LIN {X 0,Y 363.86,Z 414.069,A -85,B 0,C 180,E1 -13028.68,E2 -13028.68} C_VEL
LIN {X 0,Y 368.612,Z 450.307,A -85,B 0,C 180,E1 -13029.654,E2 -13029.654} C_VEL
LIN {X 0,Y 367.486,Z 523.043,A -85,B 0,C 180,E1 -13031.1,E2 -13031.1} C_VEL
LIN {X 0,Y 366.851,Z 536.983,A -85,B 0,C 180,E1 -13031.609,E2 -13031.609} C_VEL
LIN {X 0,Y 366.037,Z 549.991,A -85,B 0,C 180,E1 -13032.326,E2 -13032.326} C_VEL
LIN {X 0,Y 365.038,Z 561.815,A -85,B 0,C 180,E1 -13033.215,E2 -13033.215} C_VEL
LIN {X 0,Y 364.036,Z 573.232,A -85,B 0,C 180,E1 -13034.319,E2 -13034.319} C_VEL
LIN {X 0,Y 363.244,Z 583.53,A -85,B 0,C 180,E1 -13035.576,E2 -13035.576} C_VEL
LIN {X 0,Y 362.317,Z 593.595,A -85,B 0,C 180,E1 -13037.111,E2 -13037.111} C_VEL
LIN {X 0,Y 361.455,Z 602.44,A -85,B 0,C 180,E1 -13038.788,E2 -13038.788} C_VEL
LIN {X 0,Y 360.952,Z 609.493,A -85,B 0,C 180,E1 -13040.474,E2 -13040.474} C_VEL
LIN {X 0,Y 360.641,Z 615.132,A -85,B 0,C 180,E1 -13042.16,E2 -13042.16} C_VEL
LIN {X 0,Y 360.454,Z 619.728,A -85,B 0,C 180,E1 -13043.923,E2 -13043.923} C_VEL
LIN {X 0,Y 360.429,Z 622.876,A -85,B 0,C 180,E1 -13045.527,E2 -13045.527} C_VEL
LIN {X 0,Y 360.392,Z 625.76,A -85,B 0,C 180,E1 -13047.765,E2 -13047.765} C_VEL
LIN {X 0,Y 360.474,Z 626.578,A -85,B 0,C 180,E1 -13048.883,E2 -13048.883} C_VEL
LIN {X 0,Y 360.477,Z 626.96,A -85,B 0,C 180,E1 -13050,E2 -13050} C_VEL
LIN {X 0,Y 360.453,Z 626.953,A -85,B 0,C 180,E1 -13051.117,E2 -13051.117} C_VEL
LIN {X 0,Y 360.352,Z 626.554,A -85,B 0,C 180,E1 -13052.235,E2 -13052.235} C_VEL
LIN {X 0,Y 360.326,Z 625.757,A -85,B 0,C 180,E1 -13053.354,E2 -13053.354} C_VEL
LIN {X 0,Y 360.371,Z 624.522,A -85,B 0,C 180,E1 -13054.474,E2 -13054.474} C_VEL
LIN {X 0,Y 360.435,Z 622.125,A -85,B 0,C 180,E1 -13056.048,E2 -13056.048} C_VEL
LIN {X 0,Y 360.659,Z 618.313,A -85,B 0,C 180,E1 -13057.84,E2 -13057.84} C_VEL
LIN {X 0,Y 361.038,Z 613.617,A -85,B 0,C 180,E1 -13059.524,E2 -13059.524} C_VEL
LIN {X 0,Y 361.792,Z 606.572,A -85,B 0,C 180,E1 -13061.485,E2 -13061.485} C_VEL
LIN {X 0,Y 362.814,Z 598.979,A -85,B 0,C 180,E1 -13063.156,E2 -13063.156} C_VEL
LIN {X 0,Y 363.882,Z 589.935,A -85,B 0,C 180,E1 -13064.755,E2 -13064.755} C_VEL
LIN {X 0,Y 365.122,Z 579.71,A -85,B 0,C 180,E1 -13066.206,E2 -13066.206} C_VEL
LIN {X 0,Y 366.496,Z 568.849,A -85,B 0,C 180,E1 -13067.435,E2 -13067.435} C_VEL
LIN {X 0,Y 367.703,Z 558.247,A -85,B 0,C 180,E1 -13068.383,E2 -13068.383} C_VEL
LIN {X 0,Y 368.961,Z 545.524,A -85,B 0,C 180,E1 -13069.254,E2 -13069.254} C_VEL
LIN {X 0,Y 369.904,Z 532.782,A -85,B 0,C 180,E1 -13069.889,E2 -13069.889} C_VEL
LIN {X 0,Y 370.533,Z 519.302,A -85,B 0,C 180,E1 -13070.316,E2 -13070.316} C_VEL
LIN {X 0,Y 371.83,Z 449.639,A -85,B 0,C 180,E1 -13071.708,E2 -13071.708} C_VEL
LIN {X 0,Y 368.724,Z 429.89,A -85,B 0,C 180,E1 -13072.358,E2 -13072.358} C_VEL
LIN {X 0,Y 365.446,Z 413.267,A -85,B 0,C 180,E1 -13072.99,E2 -13072.99} C_VEL
LIN {X 0,Y 366.949,Z 399.466,A -85,B 0,C 180,E1 -13076.136,E2 -13076.136} C_VEL
LIN {X 0,Y 365.22,Z 390.34,A -85,B 0,C 180,E1 -13078.493,E2 -13078.493} C_VEL
LIN {X 0,Y 362.261,Z 377.933,A -85,B 0,C 180,E1 -13081.914,E2 -13081.914} C_VEL
LIN {X 0,Y 361.88,Z 376.409,A -85,B 0,C 180,E1 -13082.362,E2 -13082.362} C_VEL
LIN {X 0,Y 361.866,Z 376.411,A -85,B 0,C 180,E1 -13085.636,E2 -13085.636} C_VEL
LIN {X 0,Y 361.872,Z 376.403,A -85,B 0,C 180,E1 -13089.027,E2 -13089.027} C_VEL
LIN {X 0,Y 361.854,Z 376.402,A -85,B 0,C 180,E1 -13092.435,E2 -13092.435} C_VEL
LIN {X 0,Y 361.908,Z 376.405,A -85,B 0,C 180,E1 -13095.93,E2 -13095.93} C_VEL
LIN {X 0,Y 361.901,Z 376.405,A -85,B 0,C 180,E1 -13099.231,E2 -13099.231} C_VEL
LIN {X 0,Y 361.864,Z 376.405,A -85,B 0,C 180,E1 -13102.982,E2 -13102.982} C_VEL
LIN {X 0,Y 361.853,Z 376.404,A -85,B 0,C 180,E1 -13106.63,E2 -13106.63} C_VEL
LIN {X 0,Y 361.87,Z 376.404,A -85,B 0,C 180,E1 -13109.672,E2 -13109.672} C_VEL
LIN {X 0,Y 361.948,Z 376.394,A -85,B 0,C 180,E1 -13113.475,E2 -13113.475} C_VEL
LIN {X 0,Y 361.883,Z 376.406,A -85,B 0,C 180,E1 -13117.144,E2 -13117.144} C_VEL
LIN {X 0,Y 361.913,Z 376.402,A -85,B 0,C 180,E1 -13120.724,E2 -13120.724} C_VEL
LIN {X 0,Y 361.94,Z 376.398,A -85,B 0,C 180,E1 -13124.226,E2 -13124.226} C_VEL
LIN {X 0,Y 361.991,Z 376.389,A -85,B 0,C 180,E1 -13126.528,E2 -13126.528} C_VEL
LIN {X 0,Y 362.023,Z 376.389,A -85,B 0,C 180,E1 -13129.938,E2 -13129.938} C_VEL
LIN {X 0,Y 362.155,Z 376.365,A -85,B 0,C 180,E1 -13133.314,E2 -13133.314} C_VEL
LIN {X 0,Y 362.275,Z 376.35,A -85,B 0,C 180,E1 -13137.777,E2 -13137.777} C_VEL
LIN {X 0,Y 362.422,Z 376.339,A -85,B 0,C 180,E1 -13140,E2 -13140} C_VEL
LIN {X 0,Y 362.276,Z 376.348,A -85,B 0,C 180,E1 -13142.224,E2 -13142.224} C_VEL
LIN {X 0,Y 362.157,Z 376.369,A -85,B 0,C 180,E1 -13146.687,E2 -13146.687} C_VEL
LIN {X 0,Y 362.024,Z 376.388,A -85,B 0,C 180,E1 -13150.063,E2 -13150.063} C_VEL
LIN {X 0,Y 361.991,Z 376.393,A -85,B 0,C 180,E1 -13153.899,E2 -13153.899} C_VEL
LIN {X 0,Y 361.962,Z 376.396,A -85,B 0,C 180,E1 -13157.94,E2 -13157.94} C_VEL
LIN {X 0,Y 361.906,Z 376.404,A -85,B 0,C 180,E1 -13161.652,E2 -13161.652} C_VEL
LIN {X 0,Y 361.923,Z 376.404,A -85,B 0,C 180,E1 -13165.291,E2 -13165.291} C_VEL
LIN {X 0,Y 361.903,Z 376.402,A -85,B 0,C 180,E1 -13167.78,E2 -13167.78} C_VEL
LIN {X 0,Y 361.833,Z 376.414,A -85,B 0,C 180,E1 -13171.63,E2 -13171.63} C_VEL
LIN {X 0,Y 361.871,Z 376.401,A -85,B 0,C 180,E1 -13175.346,E2 -13175.346} C_VEL
LIN {X 0,Y 361.872,Z 376.41,A -85,B 0,C 180,E1 -13179.029,E2 -13179.029} C_VEL
LIN {X 0,Y 361.882,Z 376.4,A -85,B 0,C 180,E1 -13182.441,E2 -13182.441} C_VEL
LIN {X 0,Y 361.846,Z 376.409,A -85,B 0,C 180,E1 -13185.637,E2 -13185.637} C_VEL
LIN {X 0,Y 361.873,Z 376.574,A -85,B 0,C 180,E1 -13188.55,E2 -13188.55} C_VEL
LIN {X 0,Y 363.569,Z 383.949,A -85,B 0,C 180,E1 -13190.931,E2 -13190.931} C_VEL
LIN {X 0,Y 371.29,Z 402.274,A -85,B 0,C 180,E1 -13191.936,E2 -13191.936} C_VEL
LIN {X 0,Y 372.737,Z 408.261,A -85,B 0,C 180,E1 -13192.173,E2 -13192.173} C_VEL
LIN {X 0,Y 370.929,Z 490.598,A -85,B 0,C 180,E1 -13193.821,E2 -13193.821} C_VEL
LIN {X 0,Y 370.307,Z 504.489,A -85,B 0,C 180,E1 -13194.342,E2 -13194.342} C_VEL
LIN {X 0,Y 369.584,Z 516.079,A -85,B 0,C 180,E1 -13194.985,E2 -13194.985} C_VEL
LIN {X 0,Y 368.499,Z 528.657,A -85,B 0,C 180,E1 -13195.929,E2 -13195.929} C_VEL
LIN {X 0,Y 367.416,Z 539.356,A -85,B 0,C 180,E1 -13196.966,E2 -13196.966} C_VEL
LIN {X 0,Y 366.121,Z 550.319,A -85,B 0,C 180,E1 -13198.3,E2 -13198.3} C_VEL
LIN {X 0,Y 364.993,Z 559.126,A -85,B 0,C 180,E1 -13199.64,E2 -13199.64} C_VEL
LIN {X 0,Y 363.917,Z 567.14,A -85,B 0,C 180,E1 -13201.132,E2 -13201.132} C_VEL
LIN {X 0,Y 362.952,Z 574.158,A -85,B 0,C 180,E1 -13202.74,E2 -13202.74} C_VEL
LIN {X 0,Y 362.27,Z 579.094,A -85,B 0,C 180,E1 -13204.12,E2 -13204.12} C_VEL
LIN {X 0,Y 361.543,Z 584.472,A -85,B 0,C 180,E1 -13206.013,E2 -13206.013} C_VEL
LIN {X 0,Y 361.041,Z 588.073,A -85,B 0,C 180,E1 -13207.693,E2 -13207.693} C_VEL
LIN {X 0,Y 360.706,Z 590.795,A -85,B 0,C 180,E1 -13209.47,E2 -13209.47} C_VEL
LIN {X 0,Y 360.459,Z 592.046,A -85,B 0,C 180,E1 -13210.643,E2 -13210.643} C_VEL
LIN {X 0,Y 360.346,Z 592.816,A -85,B 0,C 180,E1 -13211.817,E2 -13211.817} C_VEL
LIN {X 0,Y 360.319,Z 593.156,A -85,B 0,C 180,E1 -13212.988,E2 -13212.988} C_VEL
LIN {X 0,Y 360.266,Z 593.094,A -85,B 0,C 180,E1 -13214.151,E2 -13214.151} C_VEL
LIN {X 0,Y 360.268,Z 592.604,A -85,B 0,C 180,E1 -13215.31,E2 -13215.31} C_VEL
LIN {X 0,Y 360.406,Z 590.903,A -85,B 0,C 180,E1 -13217.167,E2 -13217.167} C_VEL
LIN {X 0,Y 360.694,Z 587.473,A -85,B 0,C 180,E1 -13219.333,E2 -13219.333} C_VEL
LIN {X 0,Y 360.984,Z 583.589,A -85,B 0,C 180,E1 -13221.04,E2 -13221.04} C_VEL
LIN {X 0,Y 361.463,Z 578.015,A -85,B 0,C 180,E1 -13222.905,E2 -13222.905} C_VEL
LIN {X 0,Y 362.051,Z 571.018,A -85,B 0,C 180,E1 -13224.71,E2 -13224.71} C_VEL
LIN {X 0,Y 362.839,Z 562.825,A -85,B 0,C 180,E1 -13226.391,E2 -13226.391} C_VEL
LIN {X 0,Y 363.609,Z 554.46,A -85,B 0,C 180,E1 -13227.785,E2 -13227.785} C_VEL
LIN {X 0,Y 364.602,Z 544.132,A -85,B 0,C 180,E1 -13229.172,E2 -13229.172} C_VEL
LIN {X 0,Y 365.465,Z 533.637,A -85,B 0,C 180,E1 -13230.303,E2 -13230.303} C_VEL
LIN {X 0,Y 366.263,Z 522.766,A -85,B 0,C 180,E1 -13231.237,E2 -13231.237} C_VEL
LIN {X 0,Y 367.003,Z 510.308,A -85,B 0,C 180,E1 -13232.058,E2 -13232.058} C_VEL
LIN {X 0,Y 367.525,Z 497.927,A -85,B 0,C 180,E1 -13232.637,E2 -13232.637} C_VEL
LIN {X 0,Y 367.83,Z 485.609,A -85,B 0,C 180,E1 -13233.012,E2 -13233.012} C_VEL
LIN {X 0,Y 369.047,Z 405.84,A -85,B 0,C 180,E1 -13234.574,E2 -13234.574} C_VEL
LIN {X 0,Y 366.205,Z 392.374,A -85,B 0,C 180,E1 -13234.989,E2 -13234.989} C_VEL
LIN {X 0,Y 363.231,Z 382.868,A -85,B 0,C 180,E1 -13235.365,E2 -13235.365} C_VEL
LIN {X 0,Y 362.665,Z 379.195,A -85,B 0,C 180,E1 -13236.426,E2 -13236.426} C_VEL
LIN {X 0,Y 362.058,Z 377.775,A -85,B 0,C 180,E1 -13236.985,E2 -13236.985} C_VEL
LIN {X 0,Y 361.037,Z 377.05,A -85,B 0,C 180,E1 -13237.568,E2 -13237.568} C_VEL
LIN {X 0,Y 358.444,Z 376.838,A -85,B 0,C 180,E1 -13238.759,E2 -13238.759} C_VEL
LIN {X 0,Y 356.003,Z 377.137,A -85,B 0,C 180,E1 -13240.005,E2 -13240.005} C_VEL
LIN {X 0,Y 355.005,Z 377.264,A -85,B 0,C 180,E1 -13240.97,E2 -13240.97} C_VEL
LIN {X 0,Y 354.935,Z 377.274,A -85,B 0,C 180,E1 -13241.296,E2 -13241.296} C_VEL
LIN {X 0,Y 354.924,Z 377.273,A -85,B 0,C 180,E1 -13244.917,E2 -13244.917} C_VEL
LIN {X 0,Y 354.905,Z 377.273,A -85,B 0,C 180,E1 -13248.471,E2 -13248.471} C_VEL
LIN {X 0,Y 354.839,Z 377.281,A -85,B 0,C 180,E1 -13252.105,E2 -13252.105} C_VEL
LIN {X 0,Y 354.902,Z 377.274,A -85,B 0,C 180,E1 -13255.827,E2 -13255.827} C_VEL
LIN {X 0,Y 354.856,Z 377.281,A -85,B 0,C 180,E1 -13259.678,E2 -13259.678} C_VEL
LIN {X 0,Y 354.807,Z 377.286,A -85,B 0,C 180,E1 -13263.701,E2 -13263.701} C_VEL
LIN {X 0,Y 354.799,Z 377.287,A -85,B 0,C 180,E1 -13266.458,E2 -13266.458} C_VEL
LIN {X 0,Y 354.824,Z 377.286,A -85,B 0,C 180,E1 -13269.423,E2 -13269.423} C_VEL
LIN {X 0,Y 354.787,Z 377.292,A -85,B 0,C 180,E1 -13272.866,E2 -13272.866} C_VEL
LIN {X 0,Y 354.774,Z 377.289,A -85,B 0,C 180,E1 -13276.104,E2 -13276.104} C_VEL
LIN {X 0,Y 354.787,Z 377.292,A -85,B 0,C 180,E1 -13279.178,E2 -13279.178} C_VEL
LIN {X 0,Y 354.805,Z 377.287,A -85,B 0,C 180,E1 -13282.401,E2 -13282.401} C_VEL
LIN {X 0,Y 354.809,Z 377.291,A -85,B 0,C 180,E1 -13284.94,E2 -13284.94} C_VEL
LIN {X 0,Y 354.789,Z 377.289,A -85,B 0,C 180,E1 -13288.404,E2 -13288.404} C_VEL
LIN {X 0,Y 354.841,Z 377.281,A -85,B 0,C 180,E1 -13291.618,E2 -13291.618} C_VEL
LIN {X 0,Y 354.894,Z 377.275,A -85,B 0,C 180,E1 -13294.172,E2 -13294.172} C_VEL
LIN {X 0,Y 354.829,Z 377.283,A -85,B 0,C 180,E1 -13297.893,E2 -13297.893} C_VEL
LIN {X 0,Y 354.916,Z 377.272,A -85,B 0,C 180,E1 -13301.891,E2 -13301.891} C_VEL
LIN {X 0,Y 354.936,Z 377.27,A -85,B 0,C 180,E1 -13305.981,E2 -13305.981} C_VEL
LIN {X 0,Y 354.971,Z 377.265,A -85,B 0,C 180,E1 -13309.735,E2 -13309.735} C_VEL
LIN {X 0,Y 355.119,Z 377.247,A -85,B 0,C 180,E1 -13313.18,E2 -13313.18} C_VEL
LIN {X 0,Y 355.238,Z 377.232,A -85,B 0,C 180,E1 -13317.732,E2 -13317.732} C_VEL
LIN {X 0,Y 355.389,Z 377.214,A -85,B 0,C 180,E1 -13320,E2 -13320} C_VEL
LIN {X 0,Y 355.238,Z 377.235,A -85,B 0,C 180,E1 -13322.267,E2 -13322.267} C_VEL
LIN {X 0,Y 355.118,Z 377.249,A -85,B 0,C 180,E1 -13326.819,E2 -13326.819} C_VEL
LIN {X 0,Y 354.97,Z 377.27,A -85,B 0,C 180,E1 -13330.264,E2 -13330.264} C_VEL
LIN {X 0,Y 354.935,Z 377.272,A -85,B 0,C 180,E1 -13334.019,E2 -13334.019} C_VEL
LIN {X 0,Y 354.915,Z 377.276,A -85,B 0,C 180,E1 -13338.109,E2 -13338.109} C_VEL
LIN {X 0,Y 354.827,Z 377.287,A -85,B 0,C 180,E1 -13342.106,E2 -13342.106} C_VEL
LIN {X 0,Y 354.893,Z 377.277,A -85,B 0,C 180,E1 -13345.828,E2 -13345.828} C_VEL
LIN {X 0,Y 354.848,Z 377.282,A -85,B 0,C 180,E1 -13349.679,E2 -13349.679} C_VEL
LIN {X 0,Y 354.8,Z 377.288,A -85,B 0,C 180,E1 -13353.703,E2 -13353.703} C_VEL
LIN {X 0,Y 354.794,Z 377.29,A -85,B 0,C 180,E1 -13356.46,E2 -13356.46} C_VEL
LIN {X 0,Y 354.819,Z 377.284,A -85,B 0,C 180,E1 -13359.424,E2 -13359.424} C_VEL
LIN {X 0,Y 354.833,Z 377.282,A -85,B 0,C 180,E1 -13362.877,E2 -13362.877} C_VEL
LIN {X 0,Y 354.801,Z 377.291,A -85,B 0,C 180,E1 -13366.11,E2 -13366.11} C_VEL
LIN {X 0,Y 354.821,Z 377.284,A -85,B 0,C 180,E1 -13369.185,E2 -13369.185} C_VEL
LIN {X 0,Y 354.807,Z 377.287,A -85,B 0,C 180,E1 -13372.403,E2 -13372.403} C_VEL
LIN {X 0,Y 354.811,Z 377.285,A -85,B 0,C 180,E1 -13374.942,E2 -13374.942} C_VEL
LIN {X 0,Y 354.814,Z 377.286,A -85,B 0,C 180,E1 -13378.4,E2 -13378.4} C_VEL
LIN {X 0,Y 354.873,Z 377.309,A -85,B 0,C 180,E1 -13379.751,E2 -13379.751} C_VEL
LIN {X 0,Y 357.344,Z 389.276,A -85,B 0,C 180,E1 -13382.74,E2 -13382.74} C_VEL
LIN {X 0,Y 358.518,Z 396.396,A -85,B 0,C 180,E1 -13384.453,E2 -13384.453} C_VEL
LIN {X 0,Y 357.215,Z 410.591,A -85,B 0,C 180,E1 -13387.623,E2 -13387.623} C_VEL
LIN {X 0,Y 356.949,Z 413.959,A -85,B 0,C 180,E1 -13388.339,E2 -13388.339} C_VEL
LIN {X 0,Y 361.826,Z 449.698,A -85,B 0,C 180,E1 -13389.323,E2 -13389.323} C_VEL
LIN {X 0,Y 360.656,Z 522.733,A -85,B 0,C 180,E1 -13390.802,E2 -13390.802} C_VEL
LIN {X 0,Y 359.983,Z 536.659,A -85,B 0,C 180,E1 -13391.319,E2 -13391.319} C_VEL
LIN {X 0,Y 359.162,Z 549.668,A -85,B 0,C 180,E1 -13392.05,E2 -13392.05} C_VEL
LIN {X 0,Y 358.052,Z 562.287,A -85,B 0,C 180,E1 -13393.024,E2 -13393.024} C_VEL
LIN {X 0,Y 357.031,Z 573.556,A -85,B 0,C 180,E1 -13394.15,E2 -13394.15} C_VEL
LIN {X 0,Y 356.157,Z 584.466,A -85,B 0,C 180,E1 -13395.542,E2 -13395.542} C_VEL
LIN {X 0,Y 355.307,Z 592.85,A -85,B 0,C 180,E1 -13396.852,E2 -13396.852} C_VEL
LIN {X 0,Y 354.454,Z 601.776,A -85,B 0,C 180,E1 -13398.564,E2 -13398.564} C_VEL
LIN {X 0,Y 353.924,Z 608.914,A -85,B 0,C 180,E1 -13400.283,E2 -13400.283} C_VEL
LIN {X 0,Y 353.565,Z 614.604,A -85,B 0,C 180,E1 -13402.002,E2 -13402.002} C_VEL
LIN {X 0,Y 353.368,Z 619.576,A -85,B 0,C 180,E1 -13403.951,E2 -13403.951} C_VEL
LIN {X 0,Y 353.338,Z 622.437,A -85,B 0,C 180,E1 -13405.437,E2 -13405.437} C_VEL
LIN {X 0,Y 353.295,Z 625.36,A -85,B 0,C 180,E1 -13407.72,E2 -13407.72} C_VEL
LIN {X 0,Y 353.392,Z 626.212,A -85,B 0,C 180,E1 -13408.86,E2 -13408.86} C_VEL
LIN {X 0,Y 353.395,Z 626.617,A -85,B 0,C 180,E1 -13410,E2 -13410} C_VEL
LIN {X 0,Y 353.355,Z 626.626,A -85,B 0,C 180,E1 -13411.14,E2 -13411.14} C_VEL
LIN {X 0,Y 353.246,Z 625.479,A -85,B 0,C 180,E1 -13413.422,E2 -13413.422} C_VEL
LIN {X 0,Y 353.284,Z 624.273,A -85,B 0,C 180,E1 -13414.564,E2 -13414.564} C_VEL
LIN {X 0,Y 353.328,Z 622.209,A -85,B 0,C 180,E1 -13415.987,E2 -13415.987} C_VEL
LIN {X 0,Y 353.605,Z 618.147,A -85,B 0,C 180,E1 -13417.997,E2 -13417.997} C_VEL
LIN {X 0,Y 354.006,Z 613.497,A -85,B 0,C 180,E1 -13419.715,E2 -13419.715} C_VEL
LIN {X 0,Y 354.824,Z 606.503,A -85,B 0,C 180,E1 -13421.713,E2 -13421.713} C_VEL
LIN {X 0,Y 355.896,Z 598.967,A -85,B 0,C 180,E1 -13423.416,E2 -13423.416} C_VEL
LIN {X 0,Y 356.96,Z 590.321,A -85,B 0,C 180,E1 -13424.999,E2 -13424.999} C_VEL
LIN {X 0,Y 358.304,Z 579.889,A -85,B 0,C 180,E1 -13426.523,E2 -13426.523} C_VEL
LIN {X 0,Y 359.758,Z 569.166,A -85,B 0,C 180,E1 -13427.772,E2 -13427.772} C_VEL
LIN {X 0,Y 361.014,Z 558.779,A -85,B 0,C 180,E1 -13428.736,E2 -13428.736} C_VEL
LIN {X 0,Y 362.286,Z 546.334,A -85,B 0,C 180,E1 -13429.624,E2 -13429.624} C_VEL
LIN {X 0,Y 363.328,Z 533.266,A -85,B 0,C 180,E1 -13430.302,E2 -13430.302} C_VEL
LIN {X 0,Y 364.03,Z 520.256,A -85,B 0,C 180,E1 -13430.741,E2 -13430.741} C_VEL
LIN {X 0,Y 365.417,Z 450.753,A -85,B 0,C 180,E1 -13432.157,E2 -13432.157} C_VEL
LIN {X 0,Y 362.436,Z 431.394,A -85,B 0,C 180,E1 -13432.808,E2 -13432.808} C_VEL
LIN {X 0,Y 358.762,Z 412.874,A -85,B 0,C 180,E1 -13433.539,E2 -13433.539} C_VEL
LIN {X 0,Y 360.085,Z 401.05,A -85,B 0,C 180,E1 -13436.298,E2 -13436.298} C_VEL
LIN {X 0,Y 358.348,Z 391.895,A -85,B 0,C 180,E1 -13438.717,E2 -13438.717} C_VEL
LIN {X 0,Y 355.341,Z 379.317,A -85,B 0,C 180,E1 -13442.276,E2 -13442.276} C_VEL
LIN {X 0,Y 354.831,Z 377.283,A -85,B 0,C 180,E1 -13442.918,E2 -13442.918} C_VEL
LIN {X 0,Y 354.8,Z 377.291,A -85,B 0,C 180,E1 -13446.458,E2 -13446.458} C_VEL
LIN {X 0,Y 354.821,Z 377.284,A -85,B 0,C 180,E1 -13449.423,E2 -13449.423} C_VEL
LIN {X 0,Y 354.804,Z 377.283,A -85,B 0,C 180,E1 -13452.87,E2 -13452.87} C_VEL
LIN {X 0,Y 354.848,Z 377.286,A -85,B 0,C 180,E1 -13456.116,E2 -13456.116} C_VEL
LIN {X 0,Y 354.852,Z 377.283,A -85,B 0,C 180,E1 -13459.188,E2 -13459.188} C_VEL
LIN {X 0,Y 354.804,Z 377.286,A -85,B 0,C 180,E1 -13462.402,E2 -13462.402} C_VEL
LIN {X 0,Y 354.807,Z 377.287,A -85,B 0,C 180,E1 -13464.94,E2 -13464.94} C_VEL
LIN {X 0,Y 354.788,Z 377.289,A -85,B 0,C 180,E1 -13468.405,E2 -13468.405} C_VEL
LIN {X 0,Y 354.847,Z 377.283,A -85,B 0,C 180,E1 -13471.619,E2 -13471.619} C_VEL
LIN {X 0,Y 354.893,Z 377.271,A -85,B 0,C 180,E1 -13474.172,E2 -13474.172} C_VEL
LIN {X 0,Y 354.827,Z 377.278,A -85,B 0,C 180,E1 -13477.894,E2 -13477.894} C_VEL
LIN {X 0,Y 354.916,Z 377.268,A -85,B 0,C 180,E1 -13481.891,E2 -13481.891} C_VEL
LIN {X 0,Y 354.935,Z 377.27,A -85,B 0,C 180,E1 -13485.981,E2 -13485.981} C_VEL
LIN {X 0,Y 354.97,Z 377.27,A -85,B 0,C 180,E1 -13489.736,E2 -13489.736} C_VEL
LIN {X 0,Y 355.119,Z 377.24,A -85,B 0,C 180,E1 -13493.181,E2 -13493.181} C_VEL
LIN {X 0,Y 355.238,Z 377.226,A -85,B 0,C 180,E1 -13497.733,E2 -13497.733} C_VEL
LIN {X 0,Y 355.391,Z 377.215,A -85,B 0,C 180,E1 -13500,E2 -13500} C_VEL
LIN {X 0,Y 355.239,Z 377.224,A -85,B 0,C 180,E1 -13502.268,E2 -13502.268} C_VEL
LIN {X 0,Y 355.12,Z 377.244,A -85,B 0,C 180,E1 -13506.82,E2 -13506.82} C_VEL
LIN {X 0,Y 354.971,Z 377.266,A -85,B 0,C 180,E1 -13510.265,E2 -13510.265} C_VEL
LIN {X 0,Y 354.936,Z 377.271,A -85,B 0,C 180,E1 -13514.019,E2 -13514.019} C_VEL
LIN {X 0,Y 354.917,Z 377.273,A -85,B 0,C 180,E1 -13518.11,E2 -13518.11} C_VEL
LIN {X 0,Y 354.841,Z 377.283,A -85,B 0,C 180,E1 -13522.106,E2 -13522.106} C_VEL
LIN {X 0,Y 354.894,Z 377.277,A -85,B 0,C 180,E1 -13525.828,E2 -13525.828} C_VEL
LIN {X 0,Y 354.813,Z 377.285,A -85,B 0,C 180,E1 -13529.683,E2 -13529.683} C_VEL
LIN {X 0,Y 354.802,Z 377.277,A -85,B 0,C 180,E1 -13533.703,E2 -13533.703} C_VEL
LIN {X 0,Y 354.796,Z 377.291,A -85,B 0,C 180,E1 -13536.46,E2 -13536.46} C_VEL
LIN {X 0,Y 354.821,Z 377.285,A -85,B 0,C 180,E1 -13539.425,E2 -13539.425} C_VEL
LIN {X 0,Y 354.833,Z 377.281,A -85,B 0,C 180,E1 -13542.876,E2 -13542.876} C_VEL
LIN {X 0,Y 354.783,Z 377.293,A -85,B 0,C 180,E1 -13546.107,E2 -13546.107} C_VEL
LIN {X 0,Y 354.814,Z 377.389,A -85,B 0,C 180,E1 -13548.045,E2 -13548.045} C_VEL
LIN {X 0,Y 356.388,Z 384.235,A -85,B 0,C 180,E1 -13550.335,E2 -13550.335} C_VEL
LIN {X 0,Y 364.963,Z 404.134,A -85,B 0,C 180,E1 -13551.486,E2 -13551.486} C_VEL
LIN {X 0,Y 366.344,Z 409.497,A -85,B 0,C 180,E1 -13551.711,E2 -13551.711} C_VEL
LIN {X 0,Y 364.451,Z 491.149,A -85,B 0,C 180,E1 -13553.375,E2 -13553.375} C_VEL
LIN {X 0,Y 363.826,Z 504.929,A -85,B 0,C 180,E1 -13553.904,E2 -13553.904} C_VEL
LIN {X 0,Y 363.019,Z 516.869,A -85,B 0,C 180,E1 -13554.58,E2 -13554.58} C_VEL
LIN {X 0,Y 362.046,Z 527.796,A -85,B 0,C 180,E1 -13555.404,E2 -13555.404} C_VEL
LIN {X 0,Y 360.896,Z 538.696,A -85,B 0,C 180,E1 -13556.458,E2 -13556.458} C_VEL
LIN {X 0,Y 359.499,Z 549.854,A -85,B 0,C 180,E1 -13557.814,E2 -13557.814} C_VEL
LIN {X 0,Y 358.207,Z 559.688,A -85,B 0,C 180,E1 -13559.329,E2 -13559.329} C_VEL
LIN {X 0,Y 357.055,Z 567.654,A -85,B 0,C 180,E1 -13560.847,E2 -13560.847} C_VEL
LIN {X 0,Y 355.899,Z 575.485,A -85,B 0,C 180,E1 -13562.702,E2 -13562.702} C_VEL
LIN {X 0,Y 355.183,Z 580.498,A -85,B 0,C 180,E1 -13564.195,E2 -13564.195} C_VEL
LIN {X 0,Y 354.551,Z 584.755,A -85,B 0,C 180,E1 -13565.76,E2 -13565.76} C_VEL
LIN {X 0,Y 353.934,Z 589.029,A -85,B 0,C 180,E1 -13567.835,E2 -13567.835} C_VEL
LIN {X 0,Y 353.679,Z 590.826,A -85,B 0,C 180,E1 -13569.06,E2 -13569.06} C_VEL
LIN {X 0,Y 353.462,Z 592.131,A -85,B 0,C 180,E1 -13570.244,E2 -13570.244} C_VEL
LIN {X 0,Y 353.287,Z 593.034,A -85,B 0,C 180,E1 -13571.441,E2 -13571.441} C_VEL
LIN {X 0,Y 353.211,Z 593.478,A -85,B 0,C 180,E1 -13572.763,E2 -13572.763} C_VEL
LIN {X 0,Y 353.18,Z 593.076,A -85,B 0,C 180,E1 -13575.008,E2 -13575.008} C_VEL
LIN {X 0,Y 353.299,Z 591.322,A -85,B 0,C 180,E1 -13577.095,E2 -13577.095} C_VEL
LIN {X 0,Y 353.56,Z 588.282,A -85,B 0,C 180,E1 -13579.115,E2 -13579.115} C_VEL
LIN {X 0,Y 353.854,Z 584.552,A -85,B 0,C 180,E1 -13580.858,E2 -13580.858} C_VEL
LIN {X 0,Y 354.295,Z 579.422,A -85,B 0,C 180,E1 -13582.675,E2 -13582.675} C_VEL
LIN {X 0,Y 354.938,Z 572.42,A -85,B 0,C 180,E1 -13584.603,E2 -13584.603} C_VEL
LIN {X 0,Y 355.701,Z 564.458,A -85,B 0,C 180,E1 -13586.318,E2 -13586.318} C_VEL
LIN {X 0,Y 356.481,Z 556.347,A -85,B 0,C 180,E1 -13587.74,E2 -13587.74} C_VEL
LIN {X 0,Y 357.478,Z 546.435,A -85,B 0,C 180,E1 -13589.155,E2 -13589.155} C_VEL
LIN {X 0,Y 358.442,Z 535.294,A -85,B 0,C 180,E1 -13590.423,E2 -13590.423} C_VEL
LIN {X 0,Y 359.284,Z 524.404,A -85,B 0,C 180,E1 -13591.401,E2 -13591.401} C_VEL
LIN {X 0,Y 360.065,Z 512.363,A -85,B 0,C 180,E1 -13592.237,E2 -13592.237} C_VEL
LIN {X 0,Y 360.65,Z 500.013,A -85,B 0,C 180,E1 -13592.862,E2 -13592.862} C_VEL
LIN {X 0,Y 360.97,Z 487.381,A -85,B 0,C 180,E1 -13593.279,E2 -13593.279} C_VEL
LIN {X 0,Y 362.376,Z 407.238,A -85,B 0,C 180,E1 -13594.876,E2 -13594.876} C_VEL
LIN {X 0,Y 359.777,Z 394.811,A -85,B 0,C 180,E1 -13595.267,E2 -13595.267} C_VEL
LIN {X 0,Y 356.118,Z 383.178,A -85,B 0,C 180,E1 -13595.734,E2 -13595.734} C_VEL
LIN {X 0,Y 355.074,Z 377.258,A -85,B 0,C 180,E1 -13597.535,E2 -13597.535} C_VEL
LIN {X 0,Y 354.935,Z 377.274,A -85,B 0,C 180,E1 -13601.296,E2 -13601.296} C_VEL
LIN {X 0,Y 354.283,Z 377.362,A -85,B 0,C 180,E1 -13602.243,E2 -13602.243} C_VEL
LIN {X 0,Y 351.396,Z 377.719,A -85,B 0,C 180,E1 -13603.783,E2 -13603.783} C_VEL
LIN {X 0,Y 348.947,Z 378.018,A -85,B 0,C 180,E1 -13605.029,E2 -13605.029} C_VEL
LIN {X 0,Y 347.913,Z 378.145,A -85,B 0,C 180,E1 -13605.994,E2 -13605.994} C_VEL
LIN {X 0,Y 347.839,Z 378.153,A -85,B 0,C 180,E1 -13606.321,E2 -13606.321} C_VEL
LIN {X 0,Y 347.855,Z 378.153,A -85,B 0,C 180,E1 -13608.86,E2 -13608.86} C_VEL
LIN {X 0,Y 347.779,Z 378.161,A -85,B 0,C 180,E1 -13612.578,E2 -13612.578} C_VEL
LIN {X 0,Y 347.816,Z 378.161,A -85,B 0,C 180,E1 -13615.108,E2 -13615.108} C_VEL
LIN {X 0,Y 347.813,Z 378.158,A -85,B 0,C 180,E1 -13617.693,E2 -13617.693} C_VEL
LIN {X 0,Y 347.766,Z 378.162,A -85,B 0,C 180,E1 -13620.345,E2 -13620.345} C_VEL
LIN {X 0,Y 347.745,Z 378.165,A -85,B 0,C 180,E1 -13624.463,E2 -13624.463} C_VEL
LIN {X 0,Y 347.775,Z 378.161,A -85,B 0,C 180,E1 -13627.988,E2 -13627.988} C_VEL
LIN {X 0,Y 347.75,Z 378.165,A -85,B 0,C 180,E1 -13631.829,E2 -13631.829} C_VEL
LIN {X 0,Y 347.765,Z 378.169,A -85,B 0,C 180,E1 -13635.016,E2 -13635.016} C_VEL
LIN {X 0,Y 347.749,Z 378.165,A -85,B 0,C 180,E1 -13638.396,E2 -13638.396} C_VEL
LIN {X 0,Y 347.772,Z 378.162,A -85,B 0,C 180,E1 -13642.01,E2 -13642.01} C_VEL
LIN {X 0,Y 347.741,Z 378.166,A -85,B 0,C 180,E1 -13645.535,E2 -13645.535} C_VEL
LIN {X 0,Y 347.74,Z 378.167,A -85,B 0,C 180,E1 -13648.299,E2 -13648.299} C_VEL
LIN {X 0,Y 347.774,Z 378.166,A -85,B 0,C 180,E1 -13650.987,E2 -13650.987} C_VEL
LIN {X 0,Y 347.825,Z 378.155,A -85,B 0,C 180,E1 -13653.607,E2 -13653.607} C_VEL
LIN {X 0,Y 347.783,Z 378.161,A -85,B 0,C 180,E1 -13656.161,E2 -13656.161} C_VEL
LIN {X 0,Y 347.806,Z 378.157,A -85,B 0,C 180,E1 -13659.909,E2 -13659.909} C_VEL
LIN {X 0,Y 347.86,Z 378.153,A -85,B 0,C 180,E1 -13662.359,E2 -13662.359} C_VEL
LIN {X 0,Y 347.891,Z 378.147,A -85,B 0,C 180,E1 -13665.97,E2 -13665.97} C_VEL
LIN {X 0,Y 347.922,Z 378.143,A -85,B 0,C 180,E1 -13669.525,E2 -13669.525} C_VEL
LIN {X 0,Y 348.085,Z 378.125,A -85,B 0,C 180,E1 -13673.042,E2 -13673.042} C_VEL
LIN {X 0,Y 348.201,Z 378.108,A -85,B 0,C 180,E1 -13677.686,E2 -13677.686} C_VEL
LIN {X 0,Y 348.338,Z 378.092,A -85,B 0,C 180,E1 -13680,E2 -13680} C_VEL
LIN {X 0,Y 348.201,Z 378.112,A -85,B 0,C 180,E1 -13682.313,E2 -13682.313} C_VEL
LIN {X 0,Y 348.084,Z 378.124,A -85,B 0,C 180,E1 -13686.958,E2 -13686.958} C_VEL
LIN {X 0,Y 347.921,Z 378.149,A -85,B 0,C 180,E1 -13690.474,E2 -13690.474} C_VEL
LIN {X 0,Y 347.891,Z 378.151,A -85,B 0,C 180,E1 -13694.15,E2 -13694.15} C_VEL
LIN {X 0,Y 347.884,Z 378.154,A -85,B 0,C 180,E1 -13698.29,E2 -13698.29} C_VEL
LIN {X 0,Y 347.781,Z 378.161,A -85,B 0,C 180,E1 -13701.635,E2 -13701.635} C_VEL
LIN {X 0,Y 347.805,Z 378.157,A -85,B 0,C 180,E1 -13705.109,E2 -13705.109} C_VEL
LIN {X 0,Y 347.806,Z 378.159,A -85,B 0,C 180,E1 -13707.694,E2 -13707.694} C_VEL
LIN {X 0,Y 347.758,Z 378.168,A -85,B 0,C 180,E1 -13710.347,E2 -13710.347} C_VEL
LIN {X 0,Y 347.739,Z 378.169,A -85,B 0,C 180,E1 -13714.464,E2 -13714.464} C_VEL
LIN {X 0,Y 347.771,Z 378.167,A -85,B 0,C 180,E1 -13717.99,E2 -13717.99} C_VEL
LIN {X 0,Y 347.781,Z 378.164,A -85,B 0,C 180,E1 -13721.826,E2 -13721.826} C_VEL
LIN {X 0,Y 347.794,Z 378.159,A -85,B 0,C 180,E1 -13725.012,E2 -13725.012} C_VEL
LIN {X 0,Y 347.765,Z 378.165,A -85,B 0,C 180,E1 -13728.394,E2 -13728.394} C_VEL
LIN {X 0,Y 347.774,Z 378.167,A -85,B 0,C 180,E1 -13732.011,E2 -13732.011} C_VEL
LIN {X 0,Y 347.743,Z 378.168,A -85,B 0,C 180,E1 -13735.537,E2 -13735.537} C_VEL
LIN {X 0,Y 347.838,Z 378.286,A -85,B 0,C 180,E1 -13739.494,E2 -13739.494} C_VEL
LIN {X 0,Y 350.314,Z 390.14,A -85,B 0,C 180,E1 -13742.522,E2 -13742.522} C_VEL
LIN {X 0,Y 351.483,Z 396.652,A -85,B 0,C 180,E1 -13744.13,E2 -13744.13} C_VEL
LIN {X 0,Y 351.128,Z 402.43,A -85,B 0,C 180,E1 -13745.461,E2 -13745.461} C_VEL
LIN {X 0,Y 350.033,Z 413.463,A -85,B 0,C 180,E1 -13747.968,E2 -13747.968} C_VEL
LIN {X 0,Y 355.043,Z 451.237,A -85,B 0,C 180,E1 -13749.026,E2 -13749.026} C_VEL
LIN {X 0,Y 353.832,Z 522.421,A -85,B 0,C 180,E1 -13750.492,E2 -13750.492} C_VEL
LIN {X 0,Y 353.135,Z 536.339,A -85,B 0,C 180,E1 -13751.019,E2 -13751.019} C_VEL
LIN {X 0,Y 352.299,Z 549.346,A -85,B 0,C 180,E1 -13751.763,E2 -13751.763} C_VEL
LIN {X 0,Y 351.258,Z 561.17,A -85,B 0,C 180,E1 -13752.686,E2 -13752.686} C_VEL
LIN {X 0,Y 350.127,Z 572.574,A -85,B 0,C 180,E1 -13753.829,E2 -13753.829} C_VEL
LIN {X 0,Y 349.225,Z 583.278,A -85,B 0,C 180,E1 -13755.194,E2 -13755.194} C_VEL
LIN {X 0,Y 348.334,Z 592.109,A -85,B 0,C 180,E1 -13756.584,E2 -13756.584} C_VEL
LIN {X 0,Y 347.47,Z 601.106,A -85,B 0,C 180,E1 -13758.331,E2 -13758.331} C_VEL
LIN {X 0,Y 346.877,Z 608.326,A -85,B 0,C 180,E1 -13760.084,E2 -13760.084} C_VEL
LIN {X 0,Y 346.509,Z 614.07,A -85,B 0,C 180,E1 -13761.838,E2 -13761.838} C_VEL
LIN {X 0,Y 346.34,Z 618.585,A -85,B 0,C 180,E1 -13763.593,E2 -13763.593} C_VEL
LIN {X 0,Y 346.249,Z 621.993,A -85,B 0,C 180,E1 -13765.343,E2 -13765.343} C_VEL
LIN {X 0,Y 346.188,Z 623.678,A -85,B 0,C 180,E1 -13766.508,E2 -13766.508} C_VEL
LIN {X 0,Y 346.296,Z 625.836,A -85,B 0,C 180,E1 -13768.837,E2 -13768.837} C_VEL
LIN {X 0,Y 346.316,Z 626.273,A -85,B 0,C 180,E1 -13770,E2 -13770} C_VEL
LIN {X 0,Y 346.257,Z 626.301,A -85,B 0,C 180,E1 -13771.163,E2 -13771.163} C_VEL
LIN {X 0,Y 346.167,Z 625.195,A -85,B 0,C 180,E1 -13773.492,E2 -13773.492} C_VEL
LIN {X 0,Y 346.2,Z 624.024,A -85,B 0,C 180,E1 -13774.658,E2 -13774.658} C_VEL
LIN {X 0,Y 346.242,Z 622.221,A -85,B 0,C 180,E1 -13775.956,E2 -13775.956} C_VEL
LIN {X 0,Y 346.545,Z 617.973,A -85,B 0,C 180,E1 -13778.161,E2 -13778.161} C_VEL
LIN {X 0,Y 346.99,Z 613.37,A -85,B 0,C 180,E1 -13779.913,E2 -13779.913} C_VEL
LIN {X 0,Y 347.853,Z 606.442,A -85,B 0,C 180,E1 -13781.952,E2 -13781.952} C_VEL
LIN {X 0,Y 348.985,Z 598.973,A -85,B 0,C 180,E1 -13783.687,E2 -13783.687} C_VEL
LIN {X 0,Y 350.163,Z 589.978,A -85,B 0,C 180,E1 -13785.376,E2 -13785.376} C_VEL
LIN {X 0,Y 351.517,Z 580.119,A -85,B 0,C 180,E1 -13786.852,E2 -13786.852} C_VEL
LIN {X 0,Y 353.01,Z 569.513,A -85,B 0,C 180,E1 -13788.124,E2 -13788.124} C_VEL
LIN {X 0,Y 354.538,Z 557.632,A -85,B 0,C 180,E1 -13789.241,E2 -13789.241} C_VEL
LIN {X 0,Y 355.856,Z 544.949,A -85,B 0,C 180,E1 -13790.144,E2 -13790.144} C_VEL
LIN {X 0,Y 356.906,Z 532.268,A -85,B 0,C 180,E1 -13790.797,E2 -13790.797} C_VEL
LIN {X 0,Y 357.559,Z 518.674,A -85,B 0,C 180,E1 -13791.247,E2 -13791.247} C_VEL
LIN {X 0,Y 359.047,Z 451.896,A -85,B 0,C 180,E1 -13792.621,E2 -13792.621} C_VEL
LIN {X 0,Y 356.291,Z 433.71,A -85,B 0,C 180,E1 -13793.246,E2 -13793.246} C_VEL
LIN {X 0,Y 352.081,Z 412.561,A -85,B 0,C 180,E1 -13794.101,E2 -13794.101} C_VEL
LIN {X 0,Y 353.233,Z 402.71,A -85,B 0,C 180,E1 -13796.449,E2 -13796.449} C_VEL
LIN {X 0,Y 351.435,Z 393.253,A -85,B 0,C 180,E1 -13799.009,E2 -13799.009} C_VEL
LIN {X 0,Y 348.565,Z 381.278,A -85,B 0,C 180,E1 -13802.48,E2 -13802.48} C_VEL
LIN {X 0,Y 347.777,Z 378.16,A -85,B 0,C 180,E1 -13803.474,E2 -13803.474} C_VEL
LIN {X 0,Y 347.77,Z 378.167,A -85,B 0,C 180,E1 -13806.065,E2 -13806.065} C_VEL
LIN {X 0,Y 347.764,Z 378.159,A -85,B 0,C 180,E1 -13808.79,E2 -13808.79} C_VEL
LIN {X 0,Y 347.763,Z 378.156,A -85,B 0,C 180,E1 -13811.827,E2 -13811.827} C_VEL
LIN {X 0,Y 347.795,Z 378.161,A -85,B 0,C 180,E1 -13815.011,E2 -13815.011} C_VEL
LIN {X 0,Y 347.78,Z 378.165,A -85,B 0,C 180,E1 -13818.39,E2 -13818.39} C_VEL
LIN {X 0,Y 347.771,Z 378.165,A -85,B 0,C 180,E1 -13822.01,E2 -13822.01} C_VEL
LIN {X 0,Y 347.739,Z 378.168,A -85,B 0,C 180,E1 -13825.536,E2 -13825.536} C_VEL
LIN {X 0,Y 347.758,Z 378.161,A -85,B 0,C 180,E1 -13829.653,E2 -13829.653} C_VEL
LIN {X 0,Y 347.846,Z 378.152,A -85,B 0,C 180,E1 -13832.744,E2 -13832.744} C_VEL
LIN {X 0,Y 347.781,Z 378.163,A -85,B 0,C 180,E1 -13836.162,E2 -13836.162} C_VEL
LIN {X 0,Y 347.81,Z 378.162,A -85,B 0,C 180,E1 -13839.909,E2 -13839.909} C_VEL
LIN {X 0,Y 347.86,Z 378.144,A -85,B 0,C 180,E1 -13842.359,E2 -13842.359} C_VEL
LIN {X 0,Y 347.89,Z 378.147,A -85,B 0,C 180,E1 -13845.971,E2 -13845.971} C_VEL
LIN {X 0,Y 347.921,Z 378.147,A -85,B 0,C 180,E1 -13849.526,E2 -13849.526} C_VEL
LIN {X 0,Y 348.085,Z 378.115,A -85,B 0,C 180,E1 -13853.042,E2 -13853.042} C_VEL
LIN {X 0,Y 348.201,Z 378.102,A -85,B 0,C 180,E1 -13857.687,E2 -13857.687} C_VEL
LIN {X 0,Y 348.361,Z 378.091,A -85,B 0,C 180,E1 -13860,E2 -13860} C_VEL
LIN {X 0,Y 348.201,Z 378.101,A -85,B 0,C 180,E1 -13862.314,E2 -13862.314} C_VEL
LIN {X 0,Y 348.086,Z 378.119,A -85,B 0,C 180,E1 -13866.958,E2 -13866.958} C_VEL
LIN {X 0,Y 347.922,Z 378.145,A -85,B 0,C 180,E1 -13870.475,E2 -13870.475} C_VEL
LIN {X 0,Y 347.892,Z 378.149,A -85,B 0,C 180,E1 -13874.151,E2 -13874.151} C_VEL
LIN {X 0,Y 347.886,Z 378.149,A -85,B 0,C 180,E1 -13878.292,E2 -13878.292} C_VEL
LIN {X 0,Y 347.806,Z 378.16,A -85,B 0,C 180,E1 -13881.645,E2 -13881.645} C_VEL
LIN {X 0,Y 347.807,Z 378.16,A -85,B 0,C 180,E1 -13885.109,E2 -13885.109} C_VEL
LIN {X 0,Y 347.803,Z 378.158,A -85,B 0,C 180,E1 -13887.695,E2 -13887.695} C_VEL
LIN {X 0,Y 347.745,Z 378.165,A -85,B 0,C 180,E1 -13890.349,E2 -13890.349} C_VEL
LIN {X 0,Y 347.744,Z 378.154,A -85,B 0,C 180,E1 -13894.045,E2 -13894.045} C_VEL
LIN {X 0,Y 347.76,Z 378.165,A -85,B 0,C 180,E1 -13897.322,E2 -13897.322} C_VEL
LIN {X 0,Y 347.791,Z 378.162,A -85,B 0,C 180,E1 -13900.29,E2 -13900.29} C_VEL
LIN {X 0,Y 347.785,Z 378.165,A -85,B 0,C 180,E1 -13903.399,E2 -13903.399} C_VEL
LIN {X 0,Y 347.763,Z 378.163,A -85,B 0,C 180,E1 -13907.103,E2 -13907.103} C_VEL
LIN {X 0,Y 347.748,Z 378.184,A -85,B 0,C 180,E1 -13907.505,E2 -13907.505} C_VEL
LIN {X 0,Y 349.302,Z 384.722,A -85,B 0,C 180,E1 -13909.72,E2 -13909.72} C_VEL
LIN {X 0,Y 357.668,Z 403.679,A -85,B 0,C 180,E1 -13910.884,E2 -13910.884} C_VEL
LIN {X 0,Y 359.55,Z 408.856,A -85,B 0,C 180,E1 -13911.156,E2 -13911.156} C_VEL
LIN {X 0,Y 359.951,Z 411.338,A -85,B 0,C 180,E1 -13911.244,E2 -13911.244} C_VEL
LIN {X 0,Y 358.039,Z 490.46,A -85,B 0,C 180,E1 -13912.873,E2 -13912.873} C_VEL
LIN {X 0,Y 357.445,Z 503.769,A -85,B 0,C 180,E1 -13913.373,E2 -13913.373} C_VEL
LIN {X 0,Y 356.613,Z 515.73,A -85,B 0,C 180,E1 -13914.035,E2 -13914.035} C_VEL
LIN {X 0,Y 355.631,Z 526.899,A -85,B 0,C 180,E1 -13914.864,E2 -13914.864} C_VEL
LIN {X 0,Y 354.387,Z 538.056,A -85,B 0,C 180,E1 -13915.929,E2 -13915.929} C_VEL
LIN {X 0,Y 353.079,Z 548.69,A -85,B 0,C 180,E1 -13917.219,E2 -13917.219} C_VEL
LIN {X 0,Y 351.678,Z 558.504,A -85,B 0,C 180,E1 -13918.696,E2 -13918.696} C_VEL
LIN {X 0,Y 350.445,Z 566.769,A -85,B 0,C 180,E1 -13920.242,E2 -13920.242} C_VEL
LIN {X 0,Y 349.177,Z 574.815,A -85,B 0,C 180,E1 -13922.132,E2 -13922.132} C_VEL
LIN {X 0,Y 348.352,Z 580.014,A -85,B 0,C 180,E1 -13923.651,E2 -13923.651} C_VEL
LIN {X 0,Y 347.587,Z 585.024,A -85,B 0,C 180,E1 -13925.489,E2 -13925.489} C_VEL
LIN {X 0,Y 346.966,Z 588.888,A -85,B 0,C 180,E1 -13927.366,E2 -13927.366} C_VEL
LIN {X 0,Y 346.623,Z 591.131,A -85,B 0,C 180,E1 -13928.858,E2 -13928.858} C_VEL
LIN {X 0,Y 346.241,Z 593.195,A -85,B 0,C 180,E1 -13931.049,E2 -13931.049} C_VEL
LIN {X 0,Y 346.16,Z 593.805,A -85,B 0,C 180,E1 -13932.6,E2 -13932.6} C_VEL
LIN {X 0,Y 346.08,Z 593.524,A -85,B 0,C 180,E1 -13934.693,E2 -13934.693} C_VEL
LIN {X 0,Y 346.118,Z 592.799,A -85,B 0,C 180,E1 -13935.898,E2 -13935.898} C_VEL
LIN {X 0,Y 346.218,Z 591.642,A -85,B 0,C 180,E1 -13937.098,E2 -13937.098} C_VEL
LIN {X 0,Y 346.445,Z 589.09,A -85,B 0,C 180,E1 -13938.889,E2 -13938.889} C_VEL
LIN {X 0,Y 346.732,Z 585.516,A -85,B 0,C 180,E1 -13940.668,E2 -13940.668} C_VEL
LIN {X 0,Y 347.212,Z 580.093,A -85,B 0,C 180,E1 -13942.671,E2 -13942.671} C_VEL
LIN {X 0,Y 347.799,Z 573.742,A -85,B 0,C 180,E1 -13944.492,E2 -13944.492} C_VEL
LIN {X 0,Y 348.582,Z 566.079,A -85,B 0,C 180,E1 -13946.243,E2 -13946.243} C_VEL
LIN {X 0,Y 349.35,Z 558.235,A -85,B 0,C 180,E1 -13947.694,E2 -13947.694} C_VEL
LIN {X 0,Y 350.351,Z 548.629,A -85,B 0,C 180,E1 -13949.138,E2 -13949.138} C_VEL
LIN {X 0,Y 351.325,Z 537.952,A -85,B 0,C 180,E1 -13950.434,E2 -13950.434} C_VEL
LIN {X 0,Y 352.177,Z 527.705,A -85,B 0,C 180,E1 -13951.429,E2 -13951.429} C_VEL
LIN {X 0,Y 353.053,Z 515.449,A -85,B 0,C 180,E1 -13952.353,E2 -13952.353} C_VEL
LIN {X 0,Y 353.663,Z 502.633,A -85,B 0,C 180,E1 -13953.061,E2 -13953.061} C_VEL
LIN {X 0,Y 354.11,Z 489.763,A -85,B 0,C 180,E1 -13953.536,E2 -13953.536} C_VEL
LIN {X 0,Y 355.509,Z 407.695,A -85,B 0,C 180,E1 -13955.216,E2 -13955.216} C_VEL
LIN {X 0,Y 353.229,Z 396.943,A -85,B 0,C 180,E1 -13955.562,E2 -13955.562} C_VEL
LIN {X 0,Y 349.046,Z 383.533,A -85,B 0,C 180,E1 -13956.104,E2 -13956.104} C_VEL
LIN {X 0,Y 348.019,Z 378.137,A -85,B 0,C 180,E1 -13957.794,E2 -13957.794} C_VEL
LIN {X 0,Y 347.889,Z 378.15,A -85,B 0,C 180,E1 -13961.655,E2 -13961.655} C_VEL
LIN {X 0,Y 347.87,Z 378.154,A -85,B 0,C 180,E1 -13965.226,E2 -13965.226} C_VEL
LIN {X 0,Y 347.839,Z 378.153,A -85,B 0,C 180,E1 -13966.321,E2 -13966.321} C_VEL
LIN {X 0,Y 347.188,Z 378.24,A -85,B 0,C 180,E1 -13967.287,E2 -13967.287} C_VEL
LIN {X 0,Y 344.301,Z 378.596,A -85,B 0,C 180,E1 -13968.858,E2 -13968.858} C_VEL
LIN {X 0,Y 341.848,Z 378.9,A -85,B 0,C 180,E1 -13970.13,E2 -13970.13} C_VEL
LIN {X 0,Y 340.808,Z 379.033,A -85,B 0,C 180,E1 -13971.115,E2 -13971.115} C_VEL
LIN {X 0,Y 340.731,Z 379.038,A -85,B 0,C 180,E1 -13971.448,E2 -13971.448} C_VEL
LIN {X 0,Y 340.769,Z 379.036,A -85,B 0,C 180,E1 -13974.843,E2 -13974.843} C_VEL
LIN {X 0,Y 340.781,Z 379.036,A -85,B 0,C 180,E1 -13977.525,E2 -13977.525} C_VEL
LIN {X 0,Y 340.706,Z 379.047,A -85,B 0,C 180,E1 -13981.043,E2 -13981.043} C_VEL
LIN {X 0,Y 340.719,Z 379.045,A -85,B 0,C 180,E1 -13985.278,E2 -13985.278} C_VEL
LIN {X 0,Y 340.71,Z 379.042,A -85,B 0,C 180,E1 -13988.385,E2 -13988.385} C_VEL
LIN {X 0,Y 340.698,Z 379.043,A -85,B 0,C 180,E1 -13992.044,E2 -13992.044} C_VEL
LIN {X 0,Y 340.682,Z 379.047,A -85,B 0,C 180,E1 -13995.46,E2 -13995.46} C_VEL
LIN {X 0,Y 340.684,Z 379.048,A -85,B 0,C 180,E1 -13998.689,E2 -13998.689} C_VEL
LIN {X 0,Y 340.731,Z 379.039,A -85,B 0,C 180,E1 -14001.772,E2 -14001.772} C_VEL
LIN {X 0,Y 340.719,Z 379.041,A -85,B 0,C 180,E1 -14005.594,E2 -14005.594} C_VEL
LIN {X 0,Y 340.693,Z 379.048,A -85,B 0,C 180,E1 -14008.954,E2 -14008.954} C_VEL
LIN {X 0,Y 340.798,Z 379.034,A -85,B 0,C 180,E1 -14013.019,E2 -14013.019} C_VEL
LIN {X 0,Y 340.751,Z 379.036,A -85,B 0,C 180,E1 -14015.637,E2 -14015.637} C_VEL
LIN {X 0,Y 340.746,Z 379.037,A -85,B 0,C 180,E1 -14019.474,E2 -14019.474} C_VEL
LIN {X 0,Y 340.851,Z 379.024,A -85,B 0,C 180,E1 -14021.983,E2 -14021.983} C_VEL
LIN {X 0,Y 340.863,Z 379.022,A -85,B 0,C 180,E1 -14025.704,E2 -14025.704} C_VEL
LIN {X 0,Y 340.864,Z 379.023,A -85,B 0,C 180,E1 -14029.306,E2 -14029.306} C_VEL
LIN {X 0,Y 341.053,Z 379.002,A -85,B 0,C 180,E1 -14032.897,E2 -14032.897} C_VEL
LIN {X 0,Y 341.163,Z 378.985,A -85,B 0,C 180,E1 -14037.638,E2 -14037.638} C_VEL
LIN {X 0,Y 341.288,Z 378.97,A -85,B 0,C 180,E1 -14040,E2 -14040} C_VEL
LIN {X 0,Y 341.162,Z 378.989,A -85,B 0,C 180,E1 -14042.361,E2 -14042.361} C_VEL
LIN {X 0,Y 341.052,Z 378.999,A -85,B 0,C 180,E1 -14047.102,E2 -14047.102} C_VEL
LIN {X 0,Y 340.863,Z 379.025,A -85,B 0,C 180,E1 -14050.694,E2 -14050.694} C_VEL
LIN {X 0,Y 340.856,Z 379.029,A -85,B 0,C 180,E1 -14054.325,E2 -14054.325} C_VEL
LIN {X 0,Y 340.83,Z 379.031,A -85,B 0,C 180,E1 -14058.467,E2 -14058.467} C_VEL
LIN {X 0,Y 340.747,Z 379.039,A -85,B 0,C 180,E1 -14061.857,E2 -14061.857} C_VEL
LIN {X 0,Y 340.766,Z 379.035,A -85,B 0,C 180,E1 -14065.665,E2 -14065.665} C_VEL
LIN {X 0,Y 340.736,Z 379.043,A -85,B 0,C 180,E1 -14068.32,E2 -14068.32} C_VEL
LIN {X 0,Y 340.698,Z 379.043,A -85,B 0,C 180,E1 -14071.045,E2 -14071.045} C_VEL
LIN {X 0,Y 340.713,Z 379.041,A -85,B 0,C 180,E1 -14075.279,E2 -14075.279} C_VEL
LIN {X 0,Y 340.713,Z 379.044,A -85,B 0,C 180,E1 -14078.388,E2 -14078.388} C_VEL
LIN {X 0,Y 340.722,Z 379.04,A -85,B 0,C 180,E1 -14081.304,E2 -14081.304} C_VEL
LIN {X 0,Y 340.735,Z 379.04,A -85,B 0,C 180,E1 -14084.53,E2 -14084.53} C_VEL
LIN {X 0,Y 340.73,Z 379.045,A -85,B 0,C 180,E1 -14087.949,E2 -14087.949} C_VEL
LIN {X 0,Y 340.737,Z 379.042,A -85,B 0,C 180,E1 -14091.774,E2 -14091.774} C_VEL
LIN {X 0,Y 340.721,Z 379.043,A -85,B 0,C 180,E1 -14095.596,E2 -14095.596} C_VEL
LIN {X 0,Y 340.773,Z 379.111,A -85,B 0,C 180,E1 -14099.189,E2 -14099.189} C_VEL
LIN {X 0,Y 343.494,Z 392.151,A -85,B 0,C 180,E1 -14102.591,E2 -14102.591} C_VEL
LIN {X 0,Y 344.536,Z 398.843,A -85,B 0,C 180,E1 -14104.263,E2 -14104.263} C_VEL
LIN {X 0,Y 343.124,Z 413.147,A -85,B 0,C 180,E1 -14107.589,E2 -14107.589} C_VEL
LIN {X 0,Y 348.246,Z 451.861,A -85,B 0,C 180,E1 -14108.7,E2 -14108.7} C_VEL
LIN {X 0,Y 347.02,Z 521.908,A -85,B 0,C 180,E1 -14110.171,E2 -14110.171} C_VEL
LIN {X 0,Y 346.382,Z 535.137,A -85,B 0,C 180,E1 -14110.672,E2 -14110.672} C_VEL
LIN {X 0,Y 345.49,Z 547.874,A -85,B 0,C 180,E1 -14111.391,E2 -14111.391} C_VEL
LIN {X 0,Y 344.472,Z 559.997,A -85,B 0,C 180,E1 -14112.333,E2 -14112.333} C_VEL
LIN {X 0,Y 343.295,Z 571.56,A -85,B 0,C 180,E1 -14113.498,E2 -14113.498} C_VEL
LIN {X 0,Y 342.274,Z 581.902,A -85,B 0,C 180,E1 -14114.81,E2 -14114.81} C_VEL
LIN {X 0,Y 341.614,Z 589.636,A -85,B 0,C 180,E1 -14116.012,E2 -14116.012} C_VEL
LIN {X 0,Y 340.782,Z 597.647,A -85,B 0,C 180,E1 -14117.494,E2 -14117.494} C_VEL
LIN {X 0,Y 339.985,Z 605.457,A -85,B 0,C 180,E1 -14119.278,E2 -14119.278} C_VEL
LIN {X 0,Y 339.547,Z 611.721,A -85,B 0,C 180,E1 -14121.07,E2 -14121.07} C_VEL
LIN {X 0,Y 339.332,Z 616.685,A -85,B 0,C 180,E1 -14122.862,E2 -14122.862} C_VEL
LIN {X 0,Y 339.134,Z 620.227,A -85,B 0,C 180,E1 -14124.504,E2 -14124.504} C_VEL
LIN {X 0,Y 339.113,Z 623.255,A -85,B 0,C 180,E1 -14126.435,E2 -14126.435} C_VEL
LIN {X 0,Y 339.199,Z 625.453,A -85,B 0,C 180,E1 -14128.813,E2 -14128.813} C_VEL
LIN {X 0,Y 339.224,Z 625.928,A -85,B 0,C 180,E1 -14130,E2 -14130} C_VEL
LIN {X 0,Y 339.159,Z 625.975,A -85,B 0,C 180,E1 -14131.187,E2 -14131.187} C_VEL
LIN {X 0,Y 339.091,Z 624.909,A -85,B 0,C 180,E1 -14133.565,E2 -14133.565} C_VEL
LIN {X 0,Y 339.1,Z 623.777,A -85,B 0,C 180,E1 -14134.755,E2 -14134.755} C_VEL
LIN {X 0,Y 339.141,Z 622.201,A -85,B 0,C 180,E1 -14135.947,E2 -14135.947} C_VEL
LIN {X 0,Y 339.38,Z 619.063,A -85,B 0,C 180,E1 -14137.736,E2 -14137.736} C_VEL
LIN {X 0,Y 339.777,Z 614.882,A -85,B 0,C 180,E1 -14139.524,E2 -14139.524} C_VEL
LIN {X 0,Y 340.531,Z 608.535,A -85,B 0,C 180,E1 -14141.608,E2 -14141.608} C_VEL
LIN {X 0,Y 341.665,Z 601.658,A -85,B 0,C 180,E1 -14143.38,E2 -14143.38} C_VEL
LIN {X 0,Y 342.863,Z 593.108,A -85,B 0,C 180,E1 -14145.15,E2 -14145.15} C_VEL
LIN {X 0,Y 344.176,Z 584.36,A -85,B 0,C 180,E1 -14146.611,E2 -14146.611} C_VEL
LIN {X 0,Y 345.557,Z 574.797,A -85,B 0,C 180,E1 -14147.915,E2 -14147.915} C_VEL
LIN {X 0,Y 347.051,Z 564.377,A -85,B 0,C 180,E1 -14149.059,E2 -14149.059} C_VEL
LIN {X 0,Y 348.485,Z 552.943,A -85,B 0,C 180,E1 -14150.05,E2 -14150.05} C_VEL
LIN {X 0,Y 349.801,Z 539.858,A -85,B 0,C 180,E1 -14150.892,E2 -14150.892} C_VEL
LIN {X 0,Y 350.768,Z 526.717,A -85,B 0,C 180,E1 -14151.486,E2 -14151.486} C_VEL
LIN {X 0,Y 351.296,Z 513.985,A -85,B 0,C 180,E1 -14151.838,E2 -14151.838} C_VEL
LIN {X 0,Y 352.664,Z 452.503,A -85,B 0,C 180,E1 -14153.119,E2 -14153.119} C_VEL
LIN {X 0,Y 349.588,Z 432.662,A -85,B 0,C 180,E1 -14153.833,E2 -14153.833} C_VEL
LIN {X 0,Y 345.409,Z 412.127,A -85,B 0,C 180,E1 -14154.716,E2 -14154.716} C_VEL
LIN {X 0,Y 346.348,Z 404.731,A -85,B 0,C 180,E1 -14156.513,E2 -14156.513} C_VEL
LIN {X 0,Y 345.079,Z 397.225,A -85,B 0,C 180,E1 -14158.571,E2 -14158.571} C_VEL
LIN {X 0,Y 342.15,Z 384.583,A -85,B 0,C 180,E1 -14162.279,E2 -14162.279} C_VEL
LIN {X 0,Y 340.728,Z 379.042,A -85,B 0,C 180,E1 -14164.052,E2 -14164.052} C_VEL
LIN {X 0,Y 340.739,Z 379.034,A -85,B 0,C 180,E1 -14168.226,E2 -14168.226} C_VEL
LIN {X 0,Y 340.73,Z 379.031,A -85,B 0,C 180,E1 -14172.051,E2 -14172.051} C_VEL
LIN {X 0,Y 340.731,Z 379.044,A -85,B 0,C 180,E1 -14176.212,E2 -14176.212} C_VEL
LIN {X 0,Y 340.759,Z 379.037,A -85,B 0,C 180,E1 -14179.737,E2 -14179.737} C_VEL
LIN {X 0,Y 340.706,Z 379.041,A -85,B 0,C 180,E1 -14183.559,E2 -14183.559} C_VEL
LIN {X 0,Y 340.686,Z 379.041,A -85,B 0,C 180,E1 -14186.153,E2 -14186.153} C_VEL
LIN {X 0,Y 340.769,Z 379.031,A -85,B 0,C 180,E1 -14190.332,E2 -14190.332} C_VEL
LIN {X 0,Y 340.799,Z 379.031,A -85,B 0,C 180,E1 -14193.02,E2 -14193.02} C_VEL
LIN {X 0,Y 340.722,Z 379.041,A -85,B 0,C 180,E1 -14196.927,E2 -14196.927} C_VEL
LIN {X 0,Y 340.788,Z 379.034,A -85,B 0,C 180,E1 -14200.734,E2 -14200.734} C_VEL
LIN {X 0,Y 340.78,Z 379.026,A -85,B 0,C 180,E1 -14203.219,E2 -14203.219} C_VEL
LIN {X 0,Y 340.836,Z 379.023,A -85,B 0,C 180,E1 -14206.89,E2 -14206.89} C_VEL
LIN {X 0,Y 340.919,Z 379.017,A -85,B 0,C 180,E1 -14210.508,E2 -14210.508} C_VEL
LIN {X 0,Y 341.053,Z 378.99,A -85,B 0,C 180,E1 -14212.898,E2 -14212.898} C_VEL
LIN {X 0,Y 341.163,Z 378.979,A -85,B 0,C 180,E1 -14217.639,E2 -14217.639} C_VEL
LIN {X 0,Y 341.31,Z 378.969,A -85,B 0,C 180,E1 -14220,E2 -14220} C_VEL
LIN {X 0,Y 341.163,Z 378.977,A -85,B 0,C 180,E1 -14222.362,E2 -14222.362} C_VEL
LIN {X 0,Y 341.054,Z 378.994,A -85,B 0,C 180,E1 -14227.103,E2 -14227.103} C_VEL
LIN {X 0,Y 340.864,Z 379.025,A -85,B 0,C 180,E1 -14230.694,E2 -14230.694} C_VEL
LIN {X 0,Y 340.857,Z 379.025,A -85,B 0,C 180,E1 -14234.325,E2 -14234.325} C_VEL
LIN {X 0,Y 340.833,Z 379.029,A -85,B 0,C 180,E1 -14238.468,E2 -14238.468} C_VEL
LIN {X 0,Y 340.748,Z 379.039,A -85,B 0,C 180,E1 -14241.858,E2 -14241.858} C_VEL
LIN {X 0,Y 340.767,Z 379.037,A -85,B 0,C 180,E1 -14245.665,E2 -14245.665} C_VEL
LIN {X 0,Y 340.724,Z 379.041,A -85,B 0,C 180,E1 -14248.322,E2 -14248.322} C_VEL
LIN {X 0,Y 340.693,Z 379.047,A -85,B 0,C 180,E1 -14251.046,E2 -14251.046} C_VEL
LIN {X 0,Y 340.715,Z 379.034,A -85,B 0,C 180,E1 -14255.28,E2 -14255.28} C_VEL
LIN {X 0,Y 340.715,Z 379.044,A -85,B 0,C 180,E1 -14258.389,E2 -14258.389} C_VEL
LIN {X 0,Y 340.723,Z 379.04,A -85,B 0,C 180,E1 -14261.305,E2 -14261.305} C_VEL
LIN {X 0,Y 340.72,Z 379.04,A -85,B 0,C 180,E1 -14264.533,E2 -14264.533} C_VEL
LIN {X 0,Y 340.721,Z 379.06,A -85,B 0,C 180,E1 -14266.964,E2 -14266.964} C_VEL
LIN {X 0,Y 342.194,Z 385.207,A -85,B 0,C 180,E1 -14269.074,E2 -14269.074} C_VEL
LIN {X 0,Y 350.709,Z 403.974,A -85,B 0,C 180,E1 -14270.294,E2 -14270.294} C_VEL
LIN {X 0,Y 353.521,Z 411.422,A -85,B 0,C 180,E1 -14270.708,E2 -14270.708} C_VEL
LIN {X 0,Y 351.619,Z 491.803,A -85,B 0,C 180,E1 -14272.416,E2 -14272.416} C_VEL
LIN {X 0,Y 350.921,Z 505.55,A -85,B 0,C 180,E1 -14272.96,E2 -14272.96} C_VEL
LIN {X 0,Y 350.02,Z 517.781,A -85,B 0,C 180,E1 -14273.678,E2 -14273.678} C_VEL
LIN {X 0,Y 348.867,Z 529.487,A -85,B 0,C 180,E1 -14274.608,E2 -14274.608} C_VEL
LIN {X 0,Y 347.579,Z 540.372,A -85,B 0,C 180,E1 -14275.718,E2 -14275.718} C_VEL
LIN {X 0,Y 346.078,Z 551.17,A -85,B 0,C 180,E1 -14277.097,E2 -14277.097} C_VEL
LIN {X 0,Y 344.703,Z 560.498,A -85,B 0,C 180,E1 -14278.602,E2 -14278.602} C_VEL
LIN {X 0,Y 343.379,Z 568.747,A -85,B 0,C 180,E1 -14280.243,E2 -14280.243} C_VEL
LIN {X 0,Y 342.176,Z 575.979,A -85,B 0,C 180,E1 -14282.03,E2 -14282.03} C_VEL
LIN {X 0,Y 341.274,Z 581.441,A -85,B 0,C 180,E1 -14283.721,E2 -14283.721} C_VEL
LIN {X 0,Y 340.479,Z 586.264,A -85,B 0,C 180,E1 -14285.618,E2 -14285.618} C_VEL
LIN {X 0,Y 339.859,Z 589.842,A -85,B 0,C 180,E1 -14287.508,E2 -14287.508} C_VEL
LIN {X 0,Y 339.442,Z 592.31,A -85,B 0,C 180,E1 -14289.392,E2 -14289.392} C_VEL
LIN {X 0,Y 339.216,Z 593.36,A -85,B 0,C 180,E1 -14290.641,E2 -14290.641} C_VEL
LIN {X 0,Y 339.072,Z 594.138,A -85,B 0,C 180,E1 -14292.451,E2 -14292.451} C_VEL
LIN {X 0,Y 338.98,Z 593.971,A -85,B 0,C 180,E1 -14294.364,E2 -14294.364} C_VEL
LIN {X 0,Y 339.002,Z 593.316,A -85,B 0,C 180,E1 -14295.595,E2 -14295.595} C_VEL
LIN {X 0,Y 339.121,Z 592.165,A -85,B 0,C 180,E1 -14296.918,E2 -14296.918} C_VEL
LIN {X 0,Y 339.222,Z 590.76,A -85,B 0,C 180,E1 -14298.043,E2 -14298.043} C_VEL
LIN {X 0,Y 339.498,Z 587.679,A -85,B 0,C 180,E1 -14299.866,E2 -14299.866} C_VEL
LIN {X 0,Y 339.865,Z 583.528,A -85,B 0,C 180,E1 -14301.677,E2 -14301.677} C_VEL
LIN {X 0,Y 340.472,Z 577.173,A -85,B 0,C 180,E1 -14303.779,E2 -14303.779} C_VEL
LIN {X 0,Y 341.152,Z 570.267,A -85,B 0,C 180,E1 -14305.569,E2 -14305.569} C_VEL
LIN {X 0,Y 341.93,Z 563.2,A -85,B 0,C 180,E1 -14307.055,E2 -14307.055} C_VEL
LIN {X 0,Y 342.81,Z 554.685,A -85,B 0,C 180,E1 -14308.532,E2 -14308.532} C_VEL
LIN {X 0,Y 343.915,Z 544.136,A -85,B 0,C 180,E1 -14310,E2 -14310} C_VEL
LIN {X 0,Y 344.856,Z 533.707,A -85,B 0,C 180,E1 -14311.168,E2 -14311.168} C_VEL
LIN {X 0,Y 345.754,Z 522.256,A -85,B 0,C 180,E1 -14312.184,E2 -14312.184} C_VEL
LIN {X 0,Y 346.558,Z 509.124,A -85,B 0,C 180,E1 -14313.051,E2 -14313.051} C_VEL
LIN {X 0,Y 347.131,Z 495.872,A -85,B 0,C 180,E1 -14313.664,E2 -14313.664} C_VEL
LIN {X 0,Y 347.452,Z 482.825,A -85,B 0,C 180,E1 -14314.023,E2 -14314.023} C_VEL
LIN {X 0,Y 348.721,Z 408.658,A -85,B 0,C 180,E1 -14315.551,E2 -14315.551} C_VEL
LIN {X 0,Y 346.559,Z 398.568,A -85,B 0,C 180,E1 -14315.886,E2 -14315.886} C_VEL
LIN {X 0,Y 341.904,Z 383.868,A -85,B 0,C 180,E1 -14316.491,E2 -14316.491} C_VEL
LIN {X 0,Y 340.981,Z 379.013,A -85,B 0,C 180,E1 -14318.036,E2 -14318.036} C_VEL
LIN {X 0,Y 340.855,Z 379.025,A -85,B 0,C 180,E1 -14321.899,E2 -14321.899} C_VEL
LIN {X 0,Y 340.824,Z 379.031,A -85,B 0,C 180,E1 -14325.549,E2 -14325.549} C_VEL
LIN {X 0,Y 340.841,Z 379.025,A -85,B 0,C 180,E1 -14328.466,E2 -14328.466} C_VEL
LIN {X 0,Y 340.731,Z 379.038,A -85,B 0,C 180,E1 -14331.448,E2 -14331.448} C_VEL
LIN {X 0,Y 340.089,Z 379.121,A -85,B 0,C 180,E1 -14332.436,E2 -14332.436} C_VEL
LIN {X 0,Y 337.26,Z 379.475,A -85,B 0,C 180,E1 -14334.042,E2 -14334.042} C_VEL
LIN {X 0,Y 334.848,Z 379.777,A -85,B 0,C 180,E1 -14335.343,E2 -14335.343} C_VEL
LIN {X 0,Y 333.807,Z 379.901,A -85,B 0,C 180,E1 -14336.35,E2 -14336.35} C_VEL
LIN {X 0,Y 333.72,Z 379.91,A -85,B 0,C 180,E1 -14336.691,E2 -14336.691} C_VEL
LIN {X 0,Y 333.699,Z 379.915,A -85,B 0,C 180,E1 -14340.361,E2 -14340.361} C_VEL
LIN {X 0,Y 333.675,Z 379.919,A -85,B 0,C 180,E1 -14344.658,E2 -14344.658} C_VEL
LIN {X 0,Y 333.653,Z 379.922,A -85,B 0,C 180,E1 -14347.65,E2 -14347.65} C_VEL
LIN {X 0,Y 333.646,Z 379.924,A -85,B 0,C 180,E1 -14350.766,E2 -14350.766} C_VEL
LIN {X 0,Y 333.624,Z 379.924,A -85,B 0,C 180,E1 -14354.255,E2 -14354.255} C_VEL
LIN {X 0,Y 333.64,Z 379.923,A -85,B 0,C 180,E1 -14357.618,E2 -14357.618} C_VEL
LIN {X 0,Y 333.65,Z 379.924,A -85,B 0,C 180,E1 -14361.201,E2 -14361.201} C_VEL
LIN {X 0,Y 333.673,Z 379.918,A -85,B 0,C 180,E1 -14363.86,E2 -14363.86} C_VEL
LIN {X 0,Y 333.639,Z 379.923,A -85,B 0,C 180,E1 -14367.412,E2 -14367.412} C_VEL
LIN {X 0,Y 333.685,Z 379.921,A -85,B 0,C 180,E1 -14371.025,E2 -14371.025} C_VEL
LIN {X 0,Y 333.73,Z 379.911,A -85,B 0,C 180,E1 -14373.753,E2 -14373.753} C_VEL
LIN {X 0,Y 333.714,Z 379.913,A -85,B 0,C 180,E1 -14377.913,E2 -14377.913} C_VEL
LIN {X 0,Y 333.787,Z 379.904,A -85,B 0,C 180,E1 -14381.589,E2 -14381.589} C_VEL
LIN {X 0,Y 333.802,Z 379.902,A -85,B 0,C 180,E1 -14385.576,E2 -14385.576} C_VEL
LIN {X 0,Y 333.827,Z 379.9,A -85,B 0,C 180,E1 -14389.077,E2 -14389.077} C_VEL
LIN {X 0,Y 334,Z 379.882,A -85,B 0,C 180,E1 -14392.747,E2 -14392.747} C_VEL
LIN {X 0,Y 333.805,Z 379.902,A -85,B 0,C 180,E1 -14395.169,E2 -14395.169} C_VEL
LIN {X 0,Y 334.1,Z 379.864,A -85,B 0,C 180,E1 -14397.588,E2 -14397.588} C_VEL
LIN {X 0,Y 334.239,Z 379.847,A -85,B 0,C 180,E1 -14400,E2 -14400} C_VEL
LIN {X 0,Y 334.1,Z 379.867,A -85,B 0,C 180,E1 -14402.411,E2 -14402.411} C_VEL
LIN {X 0,Y 334.008,Z 379.878,A -85,B 0,C 180,E1 -14406.039,E2 -14406.039} C_VEL
LIN {X 0,Y 333.951,Z 379.889,A -85,B 0,C 180,E1 -14408.471,E2 -14408.471} C_VEL
LIN {X 0,Y 333.784,Z 379.907,A -85,B 0,C 180,E1 -14412.155,E2 -14412.155} C_VEL
LIN {X 0,Y 333.771,Z 379.908,A -85,B 0,C 180,E1 -14415.886,E2 -14415.886} C_VEL
LIN {X 0,Y 333.789,Z 379.906,A -85,B 0,C 180,E1 -14418.655,E2 -14418.655} C_VEL
LIN {X 0,Y 333.686,Z 379.922,A -85,B 0,C 180,E1 -14422.278,E2 -14422.278} C_VEL
LIN {X 0,Y 333.73,Z 379.917,A -85,B 0,C 180,E1 -14426.247,E2 -14426.247} C_VEL
LIN {X 0,Y 333.706,Z 379.914,A -85,B 0,C 180,E1 -14428.972,E2 -14428.972} C_VEL
LIN {X 0,Y 333.64,Z 379.924,A -85,B 0,C 180,E1 -14432.588,E2 -14432.588} C_VEL
LIN {X 0,Y 333.671,Z 379.924,A -85,B 0,C 180,E1 -14436.139,E2 -14436.139} C_VEL
LIN {X 0,Y 333.68,Z 379.918,A -85,B 0,C 180,E1 -14439.188,E2 -14439.188} C_VEL
LIN {X 0,Y 333.687,Z 379.918,A -85,B 0,C 180,E1 -14442.512,E2 -14442.512} C_VEL
LIN {X 0,Y 333.657,Z 379.926,A -85,B 0,C 180,E1 -14445.966,E2 -14445.966} C_VEL
LIN {X 0,Y 333.653,Z 379.921,A -85,B 0,C 180,E1 -14449.314,E2 -14449.314} C_VEL
LIN {X 0,Y 333.654,Z 379.922,A -85,B 0,C 180,E1 -14452.35,E2 -14452.35} C_VEL
LIN {X 0,Y 333.672,Z 379.92,A -85,B 0,C 180,E1 -14455.342,E2 -14455.342} C_VEL
LIN {X 0,Y 333.728,Z 380.017,A -85,B 0,C 180,E1 -14458.897,E2 -14458.897} C_VEL
LIN {X 0,Y 336.432,Z 392.864,A -85,B 0,C 180,E1 -14462.328,E2 -14462.328} C_VEL
LIN {X 0,Y 337.536,Z 399.669,A -85,B 0,C 180,E1 -14464.072,E2 -14464.072} C_VEL
LIN {X 0,Y 336.474,Z 410.37,A -85,B 0,C 180,E1 -14466.619,E2 -14466.619} C_VEL
LIN {X 0,Y 336.22,Z 412.827,A -85,B 0,C 180,E1 -14467.201,E2 -14467.201} C_VEL
LIN {X 0,Y 341.476,Z 452.864,A -85,B 0,C 180,E1 -14468.373,E2 -14468.373} C_VEL
LIN {X 0,Y 340.229,Z 521.377,A -85,B 0,C 180,E1 -14469.837,E2 -14469.837} C_VEL
LIN {X 0,Y 339.591,Z 534.677,A -85,B 0,C 180,E1 -14470.349,E2 -14470.349} C_VEL
LIN {X 0,Y 338.641,Z 547.44,A -85,B 0,C 180,E1 -14471.079,E2 -14471.079} C_VEL
LIN {X 0,Y 337.666,Z 558.794,A -85,B 0,C 180,E1 -14471.965,E2 -14471.965} C_VEL
LIN {X 0,Y 336.391,Z 570.509,A -85,B 0,C 180,E1 -14473.15,E2 -14473.15} C_VEL
LIN {X 0,Y 335.353,Z 581.276,A -85,B 0,C 180,E1 -14474.531,E2 -14474.531} C_VEL
LIN {X 0,Y 334.467,Z 590.576,A -85,B 0,C 180,E1 -14476.017,E2 -14476.017} C_VEL
LIN {X 0,Y 333.524,Z 599.725,A -85,B 0,C 180,E1 -14477.836,E2 -14477.836} C_VEL
LIN {X 0,Y 332.8,Z 607.085,A -85,B 0,C 180,E1 -14479.66,E2 -14479.66} C_VEL
LIN {X 0,Y 332.37,Z 612.97,A -85,B 0,C 180,E1 -14481.488,E2 -14481.488} C_VEL
LIN {X 0,Y 332.179,Z 617.59,A -85,B 0,C 180,E1 -14483.318,E2 -14483.318} C_VEL
LIN {X 0,Y 332.059,Z 621.085,A -85,B 0,C 180,E1 -14485.144,E2 -14485.144} C_VEL
LIN {X 0,Y 332.04,Z 622.825,A -85,B 0,C 180,E1 -14486.359,E2 -14486.359} C_VEL
LIN {X 0,Y 332.103,Z 625.065,A -85,B 0,C 180,E1 -14488.787,E2 -14488.787} C_VEL
LIN {X 0,Y 332.132,Z 625.579,A -85,B 0,C 180,E1 -14490,E2 -14490} C_VEL
LIN {X 0,Y 332.061,Z 625.65,A -85,B 0,C 180,E1 -14491.213,E2 -14491.213} C_VEL
LIN {X 0,Y 332.016,Z 624.627,A -85,B 0,C 180,E1 -14493.641,E2 -14493.641} C_VEL
LIN {X 0,Y 332.039,Z 622.328,A -85,B 0,C 180,E1 -14495.839,E2 -14495.839} C_VEL
LIN {X 0,Y 332.321,Z 618.891,A -85,B 0,C 180,E1 -14497.901,E2 -14497.901} C_VEL
LIN {X 0,Y 332.752,Z 614.759,A -85,B 0,C 180,E1 -14499.728,E2 -14499.728} C_VEL
LIN {X 0,Y 333.56,Z 608.466,A -85,B 0,C 180,E1 -14501.854,E2 -14501.854} C_VEL
LIN {X 0,Y 334.732,Z 601.648,A -85,B 0,C 180,E1 -14503.662,E2 -14503.662} C_VEL
LIN {X 0,Y 336.001,Z 593.205,A -85,B 0,C 180,E1 -14505.467,E2 -14505.467} C_VEL
LIN {X 0,Y 337.382,Z 584.554,A -85,B 0,C 180,E1 -14506.955,E2 -14506.955} C_VEL
LIN {X 0,Y 338.836,Z 575.109,A -85,B 0,C 180,E1 -14508.283,E2 -14508.283} C_VEL
LIN {X 0,Y 340.382,Z 564.84,A -85,B 0,C 180,E1 -14509.447,E2 -14509.447} C_VEL
LIN {X 0,Y 341.869,Z 553.627,A -85,B 0,C 180,E1 -14510.455,E2 -14510.455} C_VEL
LIN {X 0,Y 343.227,Z 541.014,A -85,B 0,C 180,E1 -14511.312,E2 -14511.312} C_VEL
LIN {X 0,Y 344.305,Z 527.571,A -85,B 0,C 180,E1 -14511.949,E2 -14511.949} C_VEL
LIN {X 0,Y 344.906,Z 514.221,A -85,B 0,C 180,E1 -14512.342,E2 -14512.342} C_VEL
LIN {X 0,Y 346.306,Z 453.116,A -85,B 0,C 180,E1 -14513.641,E2 -14513.641} C_VEL
LIN {X 0,Y 343.221,Z 433.407,A -85,B 0,C 180,E1 -14514.374,E2 -14514.374} C_VEL
LIN {X 0,Y 338.759,Z 411.794,A -85,B 0,C 180,E1 -14515.33,E2 -14515.33} C_VEL
LIN {X 0,Y 339.517,Z 405.721,A -85,B 0,C 180,E1 -14516.845,E2 -14516.845} C_VEL
LIN {X 0,Y 337.722,Z 396.612,A -85,B 0,C 180,E1 -14519.446,E2 -14519.446} C_VEL
LIN {X 0,Y 335.232,Z 385.996,A -85,B 0,C 180,E1 -14522.663,E2 -14522.663} C_VEL
LIN {X 0,Y 333.672,Z 379.922,A -85,B 0,C 180,E1 -14524.658,E2 -14524.658} C_VEL
LIN {X 0,Y 333.655,Z 379.92,A -85,B 0,C 180,E1 -14527.65,E2 -14527.65} C_VEL
LIN {X 0,Y 333.652,Z 379.924,A -85,B 0,C 180,E1 -14530.765,E2 -14530.765} C_VEL
LIN {X 0,Y 333.659,Z 379.925,A -85,B 0,C 180,E1 -14534.262,E2 -14534.262} C_VEL
LIN {X 0,Y 333.69,Z 379.917,A -85,B 0,C 180,E1 -14537.626,E2 -14537.626} C_VEL
LIN {X 0,Y 333.678,Z 379.919,A -85,B 0,C 180,E1 -14541.195,E2 -14541.195} C_VEL
LIN {X 0,Y 333.68,Z 379.92,A -85,B 0,C 180,E1 -14545.225,E2 -14545.225} C_VEL
LIN {X 0,Y 333.692,Z 379.913,A -85,B 0,C 180,E1 -14549.637,E2 -14549.637} C_VEL
LIN {X 0,Y 333.738,Z 379.91,A -85,B 0,C 180,E1 -14552.401,E2 -14552.401} C_VEL
LIN {X 0,Y 333.72,Z 379.91,A -85,B 0,C 180,E1 -14555.09,E2 -14555.09} C_VEL
LIN {X 0,Y 333.675,Z 379.913,A -85,B 0,C 180,E1 -14559.019,E2 -14559.019} C_VEL
LIN {X 0,Y 333.787,Z 379.903,A -85,B 0,C 180,E1 -14561.589,E2 -14561.589} C_VEL
LIN {X 0,Y 333.801,Z 379.906,A -85,B 0,C 180,E1 -14565.576,E2 -14565.576} C_VEL
LIN {X 0,Y 333.826,Z 379.898,A -85,B 0,C 180,E1 -14569.078,E2 -14569.078} C_VEL
LIN {X 0,Y 334.006,Z 379.867,A -85,B 0,C 180,E1 -14572.747,E2 -14572.747} C_VEL
LIN {X 0,Y 333.805,Z 379.906,A -85,B 0,C 180,E1 -14575.169,E2 -14575.169} C_VEL
LIN {X 0,Y 334.1,Z 379.858,A -85,B 0,C 180,E1 -14577.589,E2 -14577.589} C_VEL
LIN {X 0,Y 334.26,Z 379.847,A -85,B 0,C 180,E1 -14580,E2 -14580} C_VEL
LIN {X 0,Y 334.101,Z 379.856,A -85,B 0,C 180,E1 -14582.412,E2 -14582.412} C_VEL
LIN {X 0,Y 333.986,Z 379.873,A -85,B 0,C 180,E1 -14586.662,E2 -14586.662} C_VEL
LIN {X 0,Y 333.844,Z 379.9,A -85,B 0,C 180,E1 -14589.696,E2 -14589.696} C_VEL
LIN {X 0,Y 333.79,Z 379.906,A -85,B 0,C 180,E1 -14593.392,E2 -14593.392} C_VEL
LIN {X 0,Y 333.741,Z 379.908,A -85,B 0,C 180,E1 -14597.147,E2 -14597.147} C_VEL
LIN {X 0,Y 333.747,Z 379.906,A -85,B 0,C 180,E1 -14599.69,E2 -14599.69} C_VEL
LIN {X 0,Y 333.672,Z 379.914,A -85,B 0,C 180,E1 -14603.591,E2 -14603.591} C_VEL
LIN {X 0,Y 333.73,Z 379.914,A -85,B 0,C 180,E1 -14606.247,E2 -14606.247} C_VEL
LIN {X 0,Y 333.685,Z 379.922,A -85,B 0,C 180,E1 -14608.975,E2 -14608.975} C_VEL
LIN {X 0,Y 333.639,Z 379.924,A -85,B 0,C 180,E1 -14612.588,E2 -14612.588} C_VEL
LIN {X 0,Y 333.673,Z 379.921,A -85,B 0,C 180,E1 -14616.14,E2 -14616.14} C_VEL
LIN {X 0,Y 333.682,Z 379.92,A -85,B 0,C 180,E1 -14619.188,E2 -14619.188} C_VEL
LIN {X 0,Y 333.688,Z 379.911,A -85,B 0,C 180,E1 -14622.512,E2 -14622.512} C_VEL
LIN {X 0,Y 333.656,Z 380.017,A -85,B 0,C 180,E1 -14626.418,E2 -14626.418} C_VEL
LIN {X 0,Y 334.985,Z 385.519,A -85,B 0,C 180,E1 -14628.377,E2 -14628.377} C_VEL
LIN {X 0,Y 343.042,Z 402.709,A -85,B 0,C 180,E1 -14629.574,E2 -14629.574} C_VEL
LIN {X 0,Y 347.311,Z 412.986,A -85,B 0,C 180,E1 -14630.204,E2 -14630.204} C_VEL
LIN {X 0,Y 345.251,Z 491.971,A -85,B 0,C 180,E1 -14631.9,E2 -14631.9} C_VEL
LIN {X 0,Y 344.534,Z 505.724,A -85,B 0,C 180,E1 -14632.451,E2 -14632.451} C_VEL
LIN {X 0,Y 343.605,Z 517.831,A -85,B 0,C 180,E1 -14633.169,E2 -14633.169} C_VEL
LIN {X 0,Y 342.493,Z 528.71,A -85,B 0,C 180,E1 -14634.029,E2 -14634.029} C_VEL
LIN {X 0,Y 341.1,Z 539.983,A -85,B 0,C 180,E1 -14635.177,E2 -14635.177} C_VEL
LIN {X 0,Y 339.602,Z 550.769,A -85,B 0,C 180,E1 -14636.565,E2 -14636.565} C_VEL
LIN {X 0,Y 338.171,Z 559.752,A -85,B 0,C 180,E1 -14637.999,E2 -14637.999} C_VEL
LIN {X 0,Y 336.813,Z 567.877,A -85,B 0,C 180,E1 -14639.603,E2 -14639.603} C_VEL
LIN {X 0,Y 335.646,Z 574.546,A -85,B 0,C 180,E1 -14641.211,E2 -14641.211} C_VEL
LIN {X 0,Y 334.481,Z 580.967,A -85,B 0,C 180,E1 -14643.145,E2 -14643.145} C_VEL
LIN {X 0,Y 333.599,Z 585.973,A -85,B 0,C 180,E1 -14645.081,E2 -14645.081} C_VEL
LIN {X 0,Y 332.926,Z 589.726,A -85,B 0,C 180,E1 -14647.013,E2 -14647.013} C_VEL
LIN {X 0,Y 332.448,Z 592.348,A -85,B 0,C 180,E1 -14648.938,E2 -14648.938} C_VEL
LIN {X 0,Y 332.19,Z 593.525,A -85,B 0,C 180,E1 -14650.215,E2 -14650.215} C_VEL
LIN {X 0,Y 332.007,Z 594.468,A -85,B 0,C 180,E1 -14652.285,E2 -14652.285} C_VEL
LIN {X 0,Y 331.894,Z 594.408,A -85,B 0,C 180,E1 -14654.022,E2 -14654.022} C_VEL
LIN {X 0,Y 331.893,Z 593.831,A -85,B 0,C 180,E1 -14655.28,E2 -14655.28} C_VEL
LIN {X 0,Y 332.002,Z 592.55,A -85,B 0,C 180,E1 -14656.846,E2 -14656.846} C_VEL
LIN {X 0,Y 332.259,Z 589.6,A -85,B 0,C 180,E1 -14659.026,E2 -14659.026} C_VEL
LIN {X 0,Y 332.592,Z 585.968,A -85,B 0,C 180,E1 -14660.881,E2 -14660.881} C_VEL
LIN {X 0,Y 333.049,Z 581.21,A -85,B 0,C 180,E1 -14662.726,E2 -14662.726} C_VEL
LIN {X 0,Y 333.643,Z 575.193,A -85,B 0,C 180,E1 -14664.561,E2 -14664.561} C_VEL
LIN {X 0,Y 334.438,Z 567.703,A -85,B 0,C 180,E1 -14666.386,E2 -14666.386} C_VEL
LIN {X 0,Y 335.277,Z 560.06,A -85,B 0,C 180,E1 -14667.898,E2 -14667.898} C_VEL
LIN {X 0,Y 336.35,Z 550.764,A -85,B 0,C 180,E1 -14669.401,E2 -14669.401} C_VEL
LIN {X 0,Y 337.378,Z 540.215,A -85,B 0,C 180,E1 -14670.771,E2 -14670.771} C_VEL
LIN {X 0,Y 338.354,Z 528.979,A -85,B 0,C 180,E1 -14671.934,E2 -14671.934} C_VEL
LIN {X 0,Y 339.329,Z 516.959,A -85,B 0,C 180,E1 -14672.894,E2 -14672.894} C_VEL
LIN {X 0,Y 339.973,Z 503.718,A -85,B 0,C 180,E1 -14673.667,E2 -14673.667} C_VEL
LIN {X 0,Y 340.489,Z 490.416,A -85,B 0,C 180,E1 -14674.18,E2 -14674.18} C_VEL
LIN {X 0,Y 341.967,Z 409.612,A -85,B 0,C 180,E1 -14675.898,E2 -14675.898} C_VEL
LIN {X 0,Y 340.162,Z 401.028,A -85,B 0,C 180,E1 -14676.189,E2 -14676.189} C_VEL
LIN {X 0,Y 334.766,Z 384.208,A -85,B 0,C 180,E1 -14676.889,E2 -14676.889} C_VEL
LIN {X 0,Y 333.938,Z 379.891,A -85,B 0,C 180,E1 -14678.264,E2 -14678.264} C_VEL
LIN {X 0,Y 333.796,Z 379.904,A -85,B 0,C 180,E1 -14682.154,E2 -14682.154} C_VEL
LIN {X 0,Y 333.782,Z 379.906,A -85,B 0,C 180,E1 -14685.886,E2 -14685.886} C_VEL
LIN {X 0,Y 333.799,Z 379.903,A -85,B 0,C 180,E1 -14688.654,E2 -14688.654} C_VEL
LIN {X 0,Y 333.696,Z 379.915,A -85,B 0,C 180,E1 -14692.277,E2 -14692.277} C_VEL
LIN {X 0,Y 333.738,Z 379.91,A -85,B 0,C 180,E1 -14696.245,E2 -14696.245} C_VEL
LIN {X 0,Y 333.72,Z 379.91,A -85,B 0,C 180,E1 -14696.691,E2 -14696.691} C_VEL
LIN {X 0,Y 333.033,Z 380,A -85,B 0,C 180,E1 -14697.698,E2 -14697.698} C_VEL
LIN {X 0,Y 330.127,Z 380.365,A -85,B 0,C 180,E1 -14699.336,E2 -14699.336} C_VEL
LIN {X 0,Y 327.683,Z 380.667,A -85,B 0,C 180,E1 -14700.663,E2 -14700.663} C_VEL
LIN {X 0,Y 326.655,Z 380.794,A -85,B 0,C 180,E1 -14701.691,E2 -14701.691} C_VEL
LIN {X 0,Y 326.583,Z 380.801,A -85,B 0,C 180,E1 -14702.039,E2 -14702.039} C_VEL
LIN {X 0,Y 326.614,Z 380.799,A -85,B 0,C 180,E1 -14705.519,E2 -14705.519} C_VEL
LIN {X 0,Y 326.611,Z 380.802,A -85,B 0,C 180,E1 -14709.226,E2 -14709.226} C_VEL
LIN {X 0,Y 326.581,Z 380.806,A -85,B 0,C 180,E1 -14712.972,E2 -14712.972} C_VEL
LIN {X 0,Y 326.58,Z 380.806,A -85,B 0,C 180,E1 -14717.026,E2 -14717.026} C_VEL
LIN {X 0,Y 326.609,Z 380.802,A -85,B 0,C 180,E1 -14720.772,E2 -14720.772} C_VEL
LIN {X 0,Y 326.609,Z 380.799,A -85,B 0,C 180,E1 -14724.479,E2 -14724.479} C_VEL
LIN {X 0,Y 326.604,Z 380.799,A -85,B 0,C 180,E1 -14727.454,E2 -14727.454} C_VEL
LIN {X 0,Y 326.643,Z 380.794,A -85,B 0,C 180,E1 -14730.339,E2 -14730.339} C_VEL
LIN {X 0,Y 326.685,Z 380.791,A -85,B 0,C 180,E1 -14734.515,E2 -14734.515} C_VEL
LIN {X 0,Y 326.643,Z 380.797,A -85,B 0,C 180,E1 -14738.545,E2 -14738.545} C_VEL
LIN {X 0,Y 326.739,Z 380.783,A -85,B 0,C 180,E1 -14741.177,E2 -14741.177} C_VEL
LIN {X 0,Y 326.757,Z 380.78,A -85,B 0,C 180,E1 -14745.433,E2 -14745.433} C_VEL
LIN {X 0,Y 326.763,Z 380.782,A -85,B 0,C 180,E1 -14748.838,E2 -14748.838} C_VEL
LIN {X 0,Y 326.952,Z 380.76,A -85,B 0,C 180,E1 -14752.589,E2 -14752.589} C_VEL
LIN {X 0,Y 326.772,Z 380.779,A -85,B 0,C 180,E1 -14755.064,E2 -14755.064} C_VEL
LIN {X 0,Y 327.041,Z 380.743,A -85,B 0,C 180,E1 -14757.536,E2 -14757.536} C_VEL
LIN {X 0,Y 327.19,Z 380.724,A -85,B 0,C 180,E1 -14760,E2 -14760} C_VEL
LIN {X 0,Y 327.041,Z 380.745,A -85,B 0,C 180,E1 -14762.463,E2 -14762.463} C_VEL
LIN {X 0,Y 326.982,Z 380.754,A -85,B 0,C 180,E1 -14766.169,E2 -14766.169} C_VEL
LIN {X 0,Y 326.798,Z 380.776,A -85,B 0,C 180,E1 -14769.906,E2 -14769.906} C_VEL
LIN {X 0,Y 326.752,Z 380.781,A -85,B 0,C 180,E1 -14773.685,E2 -14773.685} C_VEL
LIN {X 0,Y 326.692,Z 380.787,A -85,B 0,C 180,E1 -14777.528,E2 -14777.528} C_VEL
LIN {X 0,Y 326.656,Z 380.796,A -85,B 0,C 180,E1 -14780.135,E2 -14780.135} C_VEL
LIN {X 0,Y 326.645,Z 380.798,A -85,B 0,C 180,E1 -14784.129,E2 -14784.129} C_VEL
LIN {X 0,Y 326.679,Z 380.79,A -85,B 0,C 180,E1 -14786.858,E2 -14786.858} C_VEL
LIN {X 0,Y 326.633,Z 380.797,A -85,B 0,C 180,E1 -14790.612,E2 -14790.612} C_VEL
LIN {X 0,Y 326.602,Z 380.804,A -85,B 0,C 180,E1 -14794.02,E2 -14794.02} C_VEL
LIN {X 0,Y 326.624,Z 380.797,A -85,B 0,C 180,E1 -14797.24,E2 -14797.24} C_VEL
LIN {X 0,Y 326.631,Z 380.801,A -85,B 0,C 180,E1 -14800.203,E2 -14800.203} C_VEL
LIN {X 0,Y 326.626,Z 380.798,A -85,B 0,C 180,E1 -14803.515,E2 -14803.515} C_VEL
LIN {X 0,Y 326.614,Z 380.798,A -85,B 0,C 180,E1 -14807.021,E2 -14807.021} C_VEL
LIN {X 0,Y 326.64,Z 380.796,A -85,B 0,C 180,E1 -14811.395,E2 -14811.395} C_VEL
LIN {X 0,Y 326.618,Z 380.798,A -85,B 0,C 180,E1 -14814.852,E2 -14814.852} C_VEL
LIN {X 0,Y 326.669,Z 380.948,A -85,B 0,C 180,E1 -14818.598,E2 -14818.598} C_VEL
LIN {X 0,Y 329.569,Z 394.753,A -85,B 0,C 180,E1 -14822.368,E2 -14822.368} C_VEL
LIN {X 0,Y 330.554,Z 401.645,A -85,B 0,C 180,E1 -14824.161,E2 -14824.161} C_VEL
LIN {X 0,Y 329.319,Z 412.495,A -85,B 0,C 180,E1 -14826.793,E2 -14826.793} C_VEL
LIN {X 0,Y 334.7,Z 452.95,A -85,B 0,C 180,E1 -14828.014,E2 -14828.014} C_VEL
LIN {X 0,Y 333.416,Z 520.808,A -85,B 0,C 180,E1 -14829.487,E2 -14829.487} C_VEL
LIN {X 0,Y 332.778,Z 534.203,A -85,B 0,C 180,E1 -14830.01,E2 -14830.01} C_VEL
LIN {X 0,Y 331.801,Z 547.005,A -85,B 0,C 180,E1 -14830.754,E2 -14830.754} C_VEL
LIN {X 0,Y 330.724,Z 559.191,A -85,B 0,C 180,E1 -14831.734,E2 -14831.734} C_VEL
LIN {X 0,Y 329.41,Z 570.771,A -85,B 0,C 180,E1 -14832.941,E2 -14832.941} C_VEL
LIN {X 0,Y 328.395,Z 580.925,A -85,B 0,C 180,E1 -14834.279,E2 -14834.279} C_VEL
LIN {X 0,Y 327.558,Z 589.788,A -85,B 0,C 180,E1 -14835.716,E2 -14835.716} C_VEL
LIN {X 0,Y 326.516,Z 599.017,A -85,B 0,C 180,E1 -14837.571,E2 -14837.571} C_VEL
LIN {X 0,Y 325.768,Z 606.444,A -85,B 0,C 180,E1 -14839.434,E2 -14839.434} C_VEL
LIN {X 0,Y 325.319,Z 612.393,A -85,B 0,C 180,E1 -14841.302,E2 -14841.302} C_VEL
LIN {X 0,Y 325.114,Z 617.072,A -85,B 0,C 180,E1 -14843.172,E2 -14843.172} C_VEL
LIN {X 0,Y 324.965,Z 620.611,A -85,B 0,C 180,E1 -14845.037,E2 -14845.037} C_VEL
LIN {X 0,Y 324.966,Z 622.393,A -85,B 0,C 180,E1 -14846.28,E2 -14846.28} C_VEL
LIN {X 0,Y 325.007,Z 624.676,A -85,B 0,C 180,E1 -14848.761,E2 -14848.761} C_VEL
LIN {X 0,Y 325.04,Z 625.221,A -85,B 0,C 180,E1 -14850,E2 -14850} C_VEL
LIN {X 0,Y 324.964,Z 625.325,A -85,B 0,C 180,E1 -14851.239,E2 -14851.239} C_VEL
LIN {X 0,Y 324.941,Z 624.345,A -85,B 0,C 180,E1 -14853.72,E2 -14853.72} C_VEL
LIN {X 0,Y 324.954,Z 622.29,A -85,B 0,C 180,E1 -14855.804,E2 -14855.804} C_VEL
LIN {X 0,Y 325.251,Z 618.719,A -85,B 0,C 180,E1 -14858.074,E2 -14858.074} C_VEL
LIN {X 0,Y 325.723,Z 614.638,A -85,B 0,C 180,E1 -14859.94,E2 -14859.94} C_VEL
LIN {X 0,Y 326.598,Z 608.408,A -85,B 0,C 180,E1 -14862.111,E2 -14862.111} C_VEL
LIN {X 0,Y 327.825,Z 601.66,A -85,B 0,C 180,E1 -14863.956,E2 -14863.956} C_VEL
LIN {X 0,Y 329.161,Z 593.324,A -85,B 0,C 180,E1 -14865.797,E2 -14865.797} C_VEL
LIN {X 0,Y 330.58,Z 584.781,A -85,B 0,C 180,E1 -14867.315,E2 -14867.315} C_VEL
LIN {X 0,Y 332.336,Z 574.278,A -85,B 0,C 180,E1 -14868.813,E2 -14868.813} C_VEL
LIN {X 0,Y 333.956,Z 563.905,A -85,B 0,C 180,E1 -14869.997,E2 -14869.997} C_VEL
LIN {X 0,Y 335.495,Z 552.548,A -85,B 0,C 180,E1 -14871.022,E2 -14871.022} C_VEL
LIN {X 0,Y 336.806,Z 540.882,A -85,B 0,C 180,E1 -14871.819,E2 -14871.819} C_VEL
LIN {X 0,Y 337.917,Z 527.526,A -85,B 0,C 180,E1 -14872.467,E2 -14872.467} C_VEL
LIN {X 0,Y 338.553,Z 514.441,A -85,B 0,C 180,E1 -14872.866,E2 -14872.866} C_VEL
LIN {X 0,Y 340.035,Z 454.17,A -85,B 0,C 180,E1 -14874.166,E2 -14874.166} C_VEL
LIN {X 0,Y 337.055,Z 435.04,A -85,B 0,C 180,E1 -14874.901,E2 -14874.901} C_VEL
LIN {X 0,Y 332.662,Z 413.872,A -85,B 0,C 180,E1 -14875.844,E2 -14875.844} C_VEL
LIN {X 0,Y 332.227,Z 411.378,A -85,B 0,C 180,E1 -14875.99,E2 -14875.99} C_VEL
LIN {X 0,Y 332.656,Z 407.997,A -85,B 0,C 180,E1 -14876.857,E2 -14876.857} C_VEL
LIN {X 0,Y 331.512,Z 401.111,A -85,B 0,C 180,E1 -14878.835,E2 -14878.835} C_VEL
LIN {X 0,Y 328.945,Z 389.848,A -85,B 0,C 180,E1 -14882.284,E2 -14882.284} C_VEL
LIN {X 0,Y 326.631,Z 380.799,A -85,B 0,C 180,E1 -14885.279,E2 -14885.279} C_VEL
LIN {X 0,Y 326.632,Z 380.793,A -85,B 0,C 180,E1 -14889.232,E2 -14889.232} C_VEL
LIN {X 0,Y 326.614,Z 380.793,A -85,B 0,C 180,E1 -14892.979,E2 -14892.979} C_VEL
LIN {X 0,Y 326.626,Z 380.799,A -85,B 0,C 180,E1 -14897.017,E2 -14897.017} C_VEL
LIN {X 0,Y 326.64,Z 380.795,A -85,B 0,C 180,E1 -14900.765,E2 -14900.765} C_VEL
LIN {X 0,Y 326.608,Z 380.801,A -85,B 0,C 180,E1 -14904.48,E2 -14904.48} C_VEL
LIN {X 0,Y 326.602,Z 380.798,A -85,B 0,C 180,E1 -14907.455,E2 -14907.455} C_VEL
LIN {X 0,Y 326.655,Z 380.788,A -85,B 0,C 180,E1 -14910.341,E2 -14910.341} C_VEL
LIN {X 0,Y 326.684,Z 380.785,A -85,B 0,C 180,E1 -14914.516,E2 -14914.516} C_VEL
LIN {X 0,Y 326.64,Z 380.788,A -85,B 0,C 180,E1 -14918.545,E2 -14918.545} C_VEL
LIN {X 0,Y 326.738,Z 380.786,A -85,B 0,C 180,E1 -14921.177,E2 -14921.177} C_VEL
LIN {X 0,Y 326.756,Z 380.785,A -85,B 0,C 180,E1 -14925.433,E2 -14925.433} C_VEL
LIN {X 0,Y 326.762,Z 380.776,A -85,B 0,C 180,E1 -14928.839,E2 -14928.839} C_VEL
LIN {X 0,Y 326.959,Z 380.744,A -85,B 0,C 180,E1 -14932.59,E2 -14932.59} C_VEL
LIN {X 0,Y 326.772,Z 380.781,A -85,B 0,C 180,E1 -14935.065,E2 -14935.065} C_VEL
LIN {X 0,Y 327.041,Z 380.737,A -85,B 0,C 180,E1 -14937.537,E2 -14937.537} C_VEL
LIN {X 0,Y 327.211,Z 380.725,A -85,B 0,C 180,E1 -14940,E2 -14940} C_VEL
LIN {X 0,Y 327.042,Z 380.735,A -85,B 0,C 180,E1 -14942.464,E2 -14942.464} C_VEL
LIN {X 0,Y 326.953,Z 380.75,A -85,B 0,C 180,E1 -14946.654,E2 -14946.654} C_VEL
LIN {X 0,Y 326.799,Z 380.776,A -85,B 0,C 180,E1 -14949.907,E2 -14949.907} C_VEL
LIN {X 0,Y 326.753,Z 380.783,A -85,B 0,C 180,E1 -14953.686,E2 -14953.686} C_VEL
LIN {X 0,Y 326.694,Z 380.79,A -85,B 0,C 180,E1 -14957.529,E2 -14957.529} C_VEL
LIN {X 0,Y 326.676,Z 380.785,A -85,B 0,C 180,E1 -14960.135,E2 -14960.135} C_VEL
LIN {X 0,Y 326.648,Z 380.788,A -85,B 0,C 180,E1 -14964.13,E2 -14964.13} C_VEL
LIN {X 0,Y 326.678,Z 380.79,A -85,B 0,C 180,E1 -14966.859,E2 -14966.859} C_VEL
LIN {X 0,Y 326.63,Z 380.796,A -85,B 0,C 180,E1 -14970.611,E2 -14970.611} C_VEL
LIN {X 0,Y 326.603,Z 380.786,A -85,B 0,C 180,E1 -14974.02,E2 -14974.02} C_VEL
LIN {X 0,Y 326.626,Z 380.798,A -85,B 0,C 180,E1 -14977.24,E2 -14977.24} C_VEL
LIN {X 0,Y 326.633,Z 380.797,A -85,B 0,C 180,E1 -14980.204,E2 -14980.204} C_VEL
LIN {X 0,Y 326.624,Z 380.801,A -85,B 0,C 180,E1 -14983.516,E2 -14983.516} C_VEL
LIN {X 0,Y 326.621,Z 380.897,A -85,B 0,C 180,E1 -14985.808,E2 -14985.808} C_VEL
LIN {X 0,Y 327.825,Z 385.894,A -85,B 0,C 180,E1 -14987.643,E2 -14987.643} C_VEL
LIN {X 0,Y 336.508,Z 403.986,A -85,B 0,C 180,E1 -14988.981,E2 -14988.981} C_VEL
LIN {X 0,Y 341.059,Z 414.899,A -85,B 0,C 180,E1 -14989.68,E2 -14989.68} C_VEL
LIN {X 0,Y 338.918,Z 492.3,A -85,B 0,C 180,E1 -14991.371,E2 -14991.371} C_VEL
LIN {X 0,Y 338.17,Z 505.876,A -85,B 0,C 180,E1 -14991.921,E2 -14991.921} C_VEL
LIN {X 0,Y 337.214,Z 518.022,A -85,B 0,C 180,E1 -14992.651,E2 -14992.651} C_VEL
LIN {X 0,Y 335.963,Z 529.624,A -85,B 0,C 180,E1 -14993.59,E2 -14993.59} C_VEL
LIN {X 0,Y 334.427,Z 541.395,A -85,B 0,C 180,E1 -14994.829,E2 -14994.829} C_VEL
LIN {X 0,Y 332.95,Z 551.494,A -85,B 0,C 180,E1 -14996.171,E2 -14996.171} C_VEL
LIN {X 0,Y 331.445,Z 560.386,A -85,B 0,C 180,E1 -14997.63,E2 -14997.63} C_VEL
LIN {X 0,Y 330.024,Z 568.458,A -85,B 0,C 180,E1 -14999.264,E2 -14999.264} C_VEL
LIN {X 0,Y 328.489,Z 576.529,A -85,B 0,C 180,E1 -15001.307,E2 -15001.307} C_VEL
LIN {X 0,Y 327.389,Z 582.411,A -85,B 0,C 180,E1 -15003.205,E2 -15003.205} C_VEL
LIN {X 0,Y 326.476,Z 587.236,A -85,B 0,C 180,E1 -15005.227,E2 -15005.227} C_VEL
LIN {X 0,Y 325.809,Z 590.661,A -85,B 0,C 180,E1 -15007.153,E2 -15007.153} C_VEL
LIN {X 0,Y 325.497,Z 592.371,A -85,B 0,C 180,E1 -15008.466,E2 -15008.466} C_VEL
LIN {X 0,Y 325.176,Z 593.646,A -85,B 0,C 180,E1 -15009.769,E2 -15009.769} C_VEL
LIN {X 0,Y 324.926,Z 594.801,A -85,B 0,C 180,E1 -15012.122,E2 -15012.122} C_VEL
LIN {X 0,Y 324.835,Z 594.787,A -85,B 0,C 180,E1 -15013.665,E2 -15013.665} C_VEL
LIN {X 0,Y 324.801,Z 594.339,A -85,B 0,C 180,E1 -15014.951,E2 -15014.951} C_VEL
LIN {X 0,Y 324.923,Z 592.959,A -85,B 0,C 180,E1 -15016.742,E2 -15016.742} C_VEL
LIN {X 0,Y 325.228,Z 589.305,A -85,B 0,C 180,E1 -15019.416,E2 -15019.416} C_VEL
LIN {X 0,Y 325.606,Z 585.464,A -85,B 0,C 180,E1 -15021.31,E2 -15021.31} C_VEL
LIN {X 0,Y 326.136,Z 580.338,A -85,B 0,C 180,E1 -15023.242,E2 -15023.242} C_VEL
LIN {X 0,Y 326.755,Z 574.225,A -85,B 0,C 180,E1 -15025.065,E2 -15025.065} C_VEL
LIN {X 0,Y 327.655,Z 566.391,A -85,B 0,C 180,E1 -15026.926,E2 -15026.926} C_VEL
LIN {X 0,Y 328.539,Z 558.391,A -85,B 0,C 180,E1 -15028.468,E2 -15028.468} C_VEL
LIN {X 0,Y 329.68,Z 548.605,A -85,B 0,C 180,E1 -15030,E2 -15030} C_VEL
LIN {X 0,Y 330.771,Z 537.736,A -85,B 0,C 180,E1 -15031.37,E2 -15031.37} C_VEL
LIN {X 0,Y 331.662,Z 527.121,A -85,B 0,C 180,E1 -15032.429,E2 -15032.429} C_VEL
LIN {X 0,Y 332.637,Z 514.318,A -85,B 0,C 180,E1 -15033.407,E2 -15033.407} C_VEL
LIN {X 0,Y 333.295,Z 502.244,A -85,B 0,C 180,E1 -15034.081,E2 -15034.081} C_VEL
LIN {X 0,Y 333.723,Z 488.871,A -85,B 0,C 180,E1 -15034.567,E2 -15034.567} C_VEL
LIN {X 0,Y 335.227,Z 410.406,A -85,B 0,C 180,E1 -15036.26,E2 -15036.26} C_VEL
LIN {X 0,Y 333.469,Z 402.463,A -85,B 0,C 180,E1 -15036.54,E2 -15036.54} C_VEL
LIN {X 0,Y 327.594,Z 384.458,A -85,B 0,C 180,E1 -15037.336,E2 -15037.336} C_VEL
LIN {X 0,Y 326.862,Z 380.772,A -85,B 0,C 180,E1 -15038.592,E2 -15038.592} C_VEL
LIN {X 0,Y 326.739,Z 380.783,A -85,B 0,C 180,E1 -15042.421,E2 -15042.421} C_VEL
LIN {X 0,Y 326.758,Z 380.782,A -85,B 0,C 180,E1 -15044.957,E2 -15044.957} C_VEL
LIN {X 0,Y 326.736,Z 380.784,A -85,B 0,C 180,E1 -15048.837,E2 -15048.837} C_VEL
LIN {X 0,Y 326.624,Z 380.798,A -85,B 0,C 180,E1 -15052.786,E2 -15052.786} C_VEL
LIN {X 0,Y 326.693,Z 380.791,A -85,B 0,C 180,E1 -15055.483,E2 -15055.483} C_VEL
LIN {X 0,Y 326.662,Z 380.793,A -85,B 0,C 180,E1 -15059.658,E2 -15059.658} C_VEL
LIN {X 0,Y 326.583,Z 380.801,A -85,B 0,C 180,E1 -15062.039,E2 -15062.039} C_VEL
LIN {X 0,Y 325.936,Z 380.887,A -85,B 0,C 180,E1 -15063.07,E2 -15063.07} C_VEL
LIN {X 0,Y 323.066,Z 381.242,A -85,B 0,C 180,E1 -15064.746,E2 -15064.746} C_VEL
LIN {X 0,Y 320.636,Z 381.542,A -85,B 0,C 180,E1 -15066.104,E2 -15066.104} C_VEL
LIN {X 0,Y 319.621,Z 381.673,A -85,B 0,C 180,E1 -15067.156,E2 -15067.156} C_VEL
LIN {X 0,Y 319.554,Z 381.677,A -85,B 0,C 180,E1 -15067.513,E2 -15067.513} C_VEL
LIN {X 0,Y 319.528,Z 381.683,A -85,B 0,C 180,E1 -15071.287,E2 -15071.287} C_VEL
LIN {X 0,Y 319.514,Z 381.685,A -85,B 0,C 180,E1 -15074.737,E2 -15074.737} C_VEL
LIN {X 0,Y 319.559,Z 381.68,A -85,B 0,C 180,E1 -15077.017,E2 -15077.017} C_VEL
LIN {X 0,Y 319.545,Z 381.679,A -85,B 0,C 180,E1 -15080.37,E2 -15080.37} C_VEL
LIN {X 0,Y 319.577,Z 381.675,A -85,B 0,C 180,E1 -15084.456,E2 -15084.456} C_VEL
LIN {X 0,Y 319.527,Z 381.68,A -85,B 0,C 180,E1 -15088.137,E2 -15088.137} C_VEL
LIN {X 0,Y 319.606,Z 381.671,A -85,B 0,C 180,E1 -15091.589,E2 -15091.589} C_VEL
LIN {X 0,Y 319.6,Z 381.671,A -85,B 0,C 180,E1 -15095.303,E2 -15095.303} C_VEL
LIN {X 0,Y 319.592,Z 381.672,A -85,B 0,C 180,E1 -15098.047,E2 -15098.047} C_VEL
LIN {X 0,Y 319.684,Z 381.664,A -85,B 0,C 180,E1 -15100.962,E2 -15100.962} C_VEL
LIN {X 0,Y 319.725,Z 381.656,A -85,B 0,C 180,E1 -15105.275,E2 -15105.275} C_VEL
LIN {X 0,Y 319.746,Z 381.652,A -85,B 0,C 180,E1 -15109.872,E2 -15109.872} C_VEL
LIN {X 0,Y 319.906,Z 381.636,A -85,B 0,C 180,E1 -15112.425,E2 -15112.425} C_VEL
LIN {X 0,Y 319.741,Z 381.655,A -85,B 0,C 180,E1 -15114.956,E2 -15114.956} C_VEL
LIN {X 0,Y 319.985,Z 381.622,A -85,B 0,C 180,E1 -15117.482,E2 -15117.482} C_VEL
LIN {X 0,Y 320.142,Z 381.601,A -85,B 0,C 180,E1 -15120,E2 -15120} C_VEL
LIN {X 0,Y 319.984,Z 381.623,A -85,B 0,C 180,E1 -15122.517,E2 -15122.517} C_VEL
LIN {X 0,Y 319.936,Z 381.632,A -85,B 0,C 180,E1 -15126.305,E2 -15126.305} C_VEL
LIN {X 0,Y 319.83,Z 381.644,A -85,B 0,C 180,E1 -15128.848,E2 -15128.848} C_VEL
LIN {X 0,Y 319.675,Z 381.664,A -85,B 0,C 180,E1 -15132.7,E2 -15132.7} C_VEL
LIN {X 0,Y 319.693,Z 381.66,A -85,B 0,C 180,E1 -15135.296,E2 -15135.296} C_VEL
LIN {X 0,Y 319.668,Z 381.662,A -85,B 0,C 180,E1 -15139.255,E2 -15139.255} C_VEL
LIN {X 0,Y 319.564,Z 381.675,A -85,B 0,C 180,E1 -15143.32,E2 -15143.32} C_VEL
LIN {X 0,Y 319.629,Z 381.672,A -85,B 0,C 180,E1 -15146.088,E2 -15146.088} C_VEL
LIN {X 0,Y 319.592,Z 381.673,A -85,B 0,C 180,E1 -15148.933,E2 -15148.933} C_VEL
LIN {X 0,Y 319.528,Z 381.683,A -85,B 0,C 180,E1 -15151.862,E2 -15151.862} C_VEL
LIN {X 0,Y 319.575,Z 381.676,A -85,B 0,C 180,E1 -15155.543,E2 -15155.543} C_VEL
LIN {X 0,Y 319.595,Z 381.678,A -85,B 0,C 180,E1 -15158.005,E2 -15158.005} C_VEL
LIN {X 0,Y 319.593,Z 381.675,A -85,B 0,C 180,E1 -15161.612,E2 -15161.612} C_VEL
LIN {X 0,Y 319.578,Z 381.675,A -85,B 0,C 180,E1 -15165.274,E2 -15165.274} C_VEL
LIN {X 0,Y 319.544,Z 381.679,A -85,B 0,C 180,E1 -15168.715,E2 -15168.715} C_VEL
LIN {X 0,Y 319.595,Z 381.674,A -85,B 0,C 180,E1 -15172.34,E2 -15172.34} C_VEL
LIN {X 0,Y 319.559,Z 381.678,A -85,B 0,C 180,E1 -15175.124,E2 -15175.124} C_VEL
LIN {X 0,Y 319.614,Z 381.81,A -85,B 0,C 180,E1 -15178.271,E2 -15178.271} C_VEL
LIN {X 0,Y 322.48,Z 395.338,A -85,B 0,C 180,E1 -15182.06,E2 -15182.06} C_VEL
LIN {X 0,Y 323.565,Z 402.316,A -85,B 0,C 180,E1 -15183.925,E2 -15183.925} C_VEL
LIN {X 0,Y 322.463,Z 412.087,A -85,B 0,C 180,E1 -15186.349,E2 -15186.349} C_VEL
LIN {X 0,Y 327.906,Z 454.504,A -85,B 0,C 180,E1 -15187.672,E2 -15187.672} C_VEL
LIN {X 0,Y 326.576,Z 521.203,A -85,B 0,C 180,E1 -15189.161,E2 -15189.161} C_VEL
LIN {X 0,Y 325.832,Z 535.107,A -85,B 0,C 180,E1 -15189.73,E2 -15189.73} C_VEL
LIN {X 0,Y 324.883,Z 547.577,A -85,B 0,C 180,E1 -15190.492,E2 -15190.492} C_VEL
LIN {X 0,Y 323.778,Z 559.52,A -85,B 0,C 180,E1 -15191.491,E2 -15191.491} C_VEL
LIN {X 0,Y 322.434,Z 570.984,A -85,B 0,C 180,E1 -15192.724,E2 -15192.724} C_VEL
LIN {X 0,Y 321.459,Z 580.557,A -85,B 0,C 180,E1 -15194.019,E2 -15194.019} C_VEL
LIN {X 0,Y 320.649,Z 588.95,A -85,B 0,C 180,E1 -15195.401,E2 -15195.401} C_VEL
LIN {X 0,Y 319.715,Z 596.909,A -85,B 0,C 180,E1 -15196.979,E2 -15196.979} C_VEL
LIN {X 0,Y 318.803,Z 604.657,A -85,B 0,C 180,E1 -15198.879,E2 -15198.879} C_VEL
LIN {X 0,Y 318.28,Z 611.808,A -85,B 0,C 180,E1 -15201.108,E2 -15201.108} C_VEL
LIN {X 0,Y 318.055,Z 616.543,A -85,B 0,C 180,E1 -15203.02,E2 -15203.02} C_VEL
LIN {X 0,Y 317.876,Z 620.131,A -85,B 0,C 180,E1 -15204.926,E2 -15204.926} C_VEL
LIN {X 0,Y 317.894,Z 621.961,A -85,B 0,C 180,E1 -15206.197,E2 -15206.197} C_VEL
LIN {X 0,Y 317.911,Z 624.287,A -85,B 0,C 180,E1 -15208.733,E2 -15208.733} C_VEL
LIN {X 0,Y 317.949,Z 624.854,A -85,B 0,C 180,E1 -15210,E2 -15210} C_VEL
LIN {X 0,Y 317.867,Z 625,A -85,B 0,C 180,E1 -15211.267,E2 -15211.267} C_VEL
LIN {X 0,Y 317.845,Z 624.064,A -85,B 0,C 180,E1 -15213.803,E2 -15213.803} C_VEL
LIN {X 0,Y 317.848,Z 622.294,A -85,B 0,C 180,E1 -15215.73,E2 -15215.73} C_VEL
LIN {X 0,Y 318.199,Z 618.551,A -85,B 0,C 180,E1 -15218.254,E2 -15218.254} C_VEL
LIN {X 0,Y 318.685,Z 614.519,A -85,B 0,C 180,E1 -15220.161,E2 -15220.161} C_VEL
LIN {X 0,Y 319.619,Z 608.363,A -85,B 0,C 180,E1 -15222.379,E2 -15222.379} C_VEL
LIN {X 0,Y 320.933,Z 601.679,A -85,B 0,C 180,E1 -15224.262,E2 -15224.262} C_VEL
LIN {X 0,Y 322.326,Z 593.471,A -85,B 0,C 180,E1 -15226.129,E2 -15226.129} C_VEL
LIN {X 0,Y 323.8,Z 584.993,A -85,B 0,C 180,E1 -15227.69,E2 -15227.69} C_VEL
LIN {X 0,Y 325.649,Z 574.618,A -85,B 0,C 180,E1 -15229.215,E2 -15229.215} C_VEL
LIN {X 0,Y 327.534,Z 562.972,A -85,B 0,C 180,E1 -15230.57,E2 -15230.57} C_VEL
LIN {X 0,Y 329.175,Z 551.43,A -85,B 0,C 180,E1 -15231.61,E2 -15231.61} C_VEL
LIN {X 0,Y 330.522,Z 539.501,A -85,B 0,C 180,E1 -15232.421,E2 -15232.421} C_VEL
LIN {X 0,Y 331.689,Z 525.743,A -85,B 0,C 180,E1 -15233.078,E2 -15233.078} C_VEL
LIN {X 0,Y 332.314,Z 513.082,A -85,B 0,C 180,E1 -15233.444,E2 -15233.444} C_VEL
LIN {X 0,Y 333.821,Z 455.431,A -85,B 0,C 180,E1 -15234.709,E2 -15234.709} C_VEL
LIN {X 0,Y 330.848,Z 436.23,A -85,B 0,C 180,E1 -15235.47,E2 -15235.47} C_VEL
LIN {X 0,Y 326.611,Z 415.72,A -85,B 0,C 180,E1 -15236.414,E2 -15236.414} C_VEL
LIN {X 0,Y 325.651,Z 411.052,A -85,B 0,C 180,E1 -15236.667,E2 -15236.667} C_VEL
LIN {X 0,Y 325.557,Z 407.197,A -85,B 0,C 180,E1 -15237.737,E2 -15237.737} C_VEL
LIN {X 0,Y 323.45,Z 397.48,A -85,B 0,C 180,E1 -15240.704,E2 -15240.704} C_VEL
LIN {X 0,Y 321.215,Z 388.064,A -85,B 0,C 180,E1 -15243.755,E2 -15243.755} C_VEL
LIN {X 0,Y 319.566,Z 381.679,A -85,B 0,C 180,E1 -15245.99,E2 -15245.99} C_VEL
LIN {X 0,Y 319.562,Z 381.678,A -85,B 0,C 180,E1 -15249.669,E2 -15249.669} C_VEL
LIN {X 0,Y 319.585,Z 381.673,A -85,B 0,C 180,E1 -15253.473,E2 -15253.473} C_VEL
LIN {X 0,Y 319.602,Z 381.674,A -85,B 0,C 180,E1 -15257.025,E2 -15257.025} C_VEL
LIN {X 0,Y 319.581,Z 381.673,A -85,B 0,C 180,E1 -15260.376,E2 -15260.376} C_VEL
LIN {X 0,Y 319.555,Z 381.675,A -85,B 0,C 180,E1 -15263.572,E2 -15263.572} C_VEL
LIN {X 0,Y 319.572,Z 381.67,A -85,B 0,C 180,E1 -15266.686,E2 -15266.686} C_VEL
LIN {X 0,Y 319.586,Z 381.669,A -85,B 0,C 180,E1 -15269.616,E2 -15269.616} C_VEL
LIN {X 0,Y 319.603,Z 381.671,A -85,B 0,C 180,E1 -15272.498,E2 -15272.498} C_VEL
LIN {X 0,Y 319.598,Z 381.671,A -85,B 0,C 180,E1 -15275.304,E2 -15275.304} C_VEL
LIN {X 0,Y 319.59,Z 381.665,A -85,B 0,C 180,E1 -15278.047,E2 -15278.047} C_VEL
LIN {X 0,Y 319.683,Z 381.664,A -85,B 0,C 180,E1 -15280.962,E2 -15280.962} C_VEL
LIN {X 0,Y 319.724,Z 381.66,A -85,B 0,C 180,E1 -15285.276,E2 -15285.276} C_VEL
LIN {X 0,Y 319.75,Z 381.656,A -85,B 0,C 180,E1 -15289.873,E2 -15289.873} C_VEL
LIN {X 0,Y 319.918,Z 381.621,A -85,B 0,C 180,E1 -15292.426,E2 -15292.426} C_VEL
LIN {X 0,Y 319.741,Z 381.656,A -85,B 0,C 180,E1 -15294.956,E2 -15294.956} C_VEL
LIN {X 0,Y 319.985,Z 381.616,A -85,B 0,C 180,E1 -15297.483,E2 -15297.483} C_VEL
LIN {X 0,Y 320.162,Z 381.604,A -85,B 0,C 180,E1 -15300,E2 -15300} C_VEL
LIN {X 0,Y 319.985,Z 381.614,A -85,B 0,C 180,E1 -15302.518,E2 -15302.518} C_VEL
LIN {X 0,Y 319.914,Z 381.627,A -85,B 0,C 180,E1 -15306.642,E2 -15306.642} C_VEL
LIN {X 0,Y 319.746,Z 381.655,A -85,B 0,C 180,E1 -15310.128,E2 -15310.128} C_VEL
LIN {X 0,Y 319.725,Z 381.66,A -85,B 0,C 180,E1 -15314.725,E2 -15314.725} C_VEL
LIN {X 0,Y 319.686,Z 381.662,A -85,B 0,C 180,E1 -15319.04,E2 -15319.04} C_VEL
LIN {X 0,Y 319.566,Z 381.673,A -85,B 0,C 180,E1 -15323.32,E2 -15323.32} C_VEL
LIN {X 0,Y 319.629,Z 381.67,A -85,B 0,C 180,E1 -15326.089,E2 -15326.089} C_VEL
LIN {X 0,Y 319.576,Z 381.68,A -85,B 0,C 180,E1 -15328.935,E2 -15328.935} C_VEL
LIN {X 0,Y 319.526,Z 381.685,A -85,B 0,C 180,E1 -15331.863,E2 -15331.863} C_VEL
LIN {X 0,Y 319.577,Z 381.669,A -85,B 0,C 180,E1 -15335.544,E2 -15335.544} C_VEL
LIN {X 0,Y 319.581,Z 381.674,A -85,B 0,C 180,E1 -15338.008,E2 -15338.008} C_VEL
LIN {X 0,Y 319.595,Z 381.668,A -85,B 0,C 180,E1 -15341.612,E2 -15341.612} C_VEL
LIN {X 0,Y 319.566,Z 381.765,A -85,B 0,C 180,E1 -15345.162,E2 -15345.162} C_VEL
LIN {X 0,Y 320.638,Z 386.191,A -85,B 0,C 180,E1 -15346.863,E2 -15346.863} C_VEL
LIN {X 0,Y 329.838,Z 404.996,A -85,B 0,C 180,E1 -15348.34,E2 -15348.34} C_VEL
LIN {X 0,Y 334.832,Z 416.844,A -85,B 0,C 180,E1 -15349.133,E2 -15349.133} C_VEL
LIN {X 0,Y 332.645,Z 492.214,A -85,B 0,C 180,E1 -15350.802,E2 -15350.802} C_VEL
LIN {X 0,Y 331.884,Z 505.914,A -85,B 0,C 180,E1 -15351.363,E2 -15351.363} C_VEL
LIN {X 0,Y 330.892,Z 517.757,A -85,B 0,C 180,E1 -15352.077,E2 -15352.077} C_VEL
LIN {X 0,Y 329.675,Z 528.878,A -85,B 0,C 180,E1 -15352.971,E2 -15352.971} C_VEL
LIN {X 0,Y 328.158,Z 540.008,A -85,B 0,C 180,E1 -15354.127,E2 -15354.127} C_VEL
LIN {X 0,Y 326.471,Z 551.086,A -85,B 0,C 180,E1 -15355.593,E2 -15355.593} C_VEL
LIN {X 0,Y 324.74,Z 561.017,A -85,B 0,C 180,E1 -15357.246,E2 -15357.246} C_VEL
LIN {X 0,Y 323.245,Z 569.038,A -85,B 0,C 180,E1 -15358.911,E2 -15358.911} C_VEL
LIN {X 0,Y 321.673,Z 576.807,A -85,B 0,C 180,E1 -15360.92,E2 -15360.92} C_VEL
LIN {X 0,Y 320.637,Z 581.962,A -85,B 0,C 180,E1 -15362.594,E2 -15362.594} C_VEL
LIN {X 0,Y 319.593,Z 587.279,A -85,B 0,C 180,E1 -15364.79,E2 -15364.79} C_VEL
LIN {X 0,Y 318.902,Z 590.583,A -85,B 0,C 180,E1 -15366.629,E2 -15366.629} C_VEL
LIN {X 0,Y 318.523,Z 592.4,A -85,B 0,C 180,E1 -15367.97,E2 -15367.97} C_VEL
LIN {X 0,Y 318.196,Z 593.746,A -85,B 0,C 180,E1 -15369.306,E2 -15369.306} C_VEL
LIN {X 0,Y 317.963,Z 594.669,A -85,B 0,C 180,E1 -15370.638,E2 -15370.638} C_VEL
LIN {X 0,Y 317.859,Z 595.136,A -85,B 0,C 180,E1 -15371.969,E2 -15371.969} C_VEL
LIN {X 0,Y 317.762,Z 595.163,A -85,B 0,C 180,E1 -15373.291,E2 -15373.291} C_VEL
LIN {X 0,Y 317.717,Z 594.788,A -85,B 0,C 180,E1 -15374.607,E2 -15374.607} C_VEL
LIN {X 0,Y 317.822,Z 593.348,A -85,B 0,C 180,E1 -15376.651,E2 -15376.651} C_VEL
LIN {X 0,Y 318.11,Z 590.09,A -85,B 0,C 180,E1 -15379.176,E2 -15379.176} C_VEL
LIN {X 0,Y 318.482,Z 586.396,A -85,B 0,C 180,E1 -15381.114,E2 -15381.114} C_VEL
LIN {X 0,Y 319.063,Z 580.824,A -85,B 0,C 180,E1 -15383.301,E2 -15383.301} C_VEL
LIN {X 0,Y 319.765,Z 574.355,A -85,B 0,C 180,E1 -15385.272,E2 -15385.272} C_VEL
LIN {X 0,Y 320.677,Z 566.461,A -85,B 0,C 180,E1 -15387.174,E2 -15387.174} C_VEL
LIN {X 0,Y 321.602,Z 558.408,A -85,B 0,C 180,E1 -15388.748,E2 -15388.748} C_VEL
LIN {X 0,Y 322.782,Z 548.558,A -85,B 0,C 180,E1 -15390.312,E2 -15390.312} C_VEL
LIN {X 0,Y 323.906,Z 537.916,A -85,B 0,C 180,E1 -15391.671,E2 -15391.671} C_VEL
LIN {X 0,Y 324.851,Z 526.829,A -85,B 0,C 180,E1 -15392.79,E2 -15392.79} C_VEL
LIN {X 0,Y 325.788,Z 514.978,A -85,B 0,C 180,E1 -15393.711,E2 -15393.711} C_VEL
LIN {X 0,Y 326.526,Z 502.242,A -85,B 0,C 180,E1 -15394.436,E2 -15394.436} C_VEL
LIN {X 0,Y 326.937,Z 490.042,A -85,B 0,C 180,E1 -15394.894,E2 -15394.894} C_VEL
LIN {X 0,Y 328.568,Z 411.629,A -85,B 0,C 180,E1 -15396.618,E2 -15396.618} C_VEL
LIN {X 0,Y 326.814,Z 404.103,A -85,B 0,C 180,E1 -15396.895,E2 -15396.895} C_VEL
LIN {X 0,Y 320.48,Z 384.903,A -85,B 0,C 180,E1 -15397.745,E2 -15397.745} C_VEL
LIN {X 0,Y 319.825,Z 381.648,A -85,B 0,C 180,E1 -15398.848,E2 -15398.848} C_VEL
LIN {X 0,Y 319.687,Z 381.663,A -85,B 0,C 180,E1 -15402.699,E2 -15402.699} C_VEL
LIN {X 0,Y 319.704,Z 381.664,A -85,B 0,C 180,E1 -15405.295,E2 -15405.295} C_VEL
LIN {X 0,Y 319.678,Z 381.667,A -85,B 0,C 180,E1 -15409.254,E2 -15409.254} C_VEL
LIN {X 0,Y 319.574,Z 381.678,A -85,B 0,C 180,E1 -15413.319,E2 -15413.319} C_VEL
LIN {X 0,Y 319.637,Z 381.667,A -85,B 0,C 180,E1 -15416.087,E2 -15416.087} C_VEL
LIN {X 0,Y 319.592,Z 381.675,A -85,B 0,C 180,E1 -15418.933,E2 -15418.933} C_VEL
LIN {X 0,Y 319.53,Z 381.679,A -85,B 0,C 180,E1 -15422.034,E2 -15422.034} C_VEL
LIN {X 0,Y 319.581,Z 381.675,A -85,B 0,C 180,E1 -15425.542,E2 -15425.542} C_VEL
LIN {X 0,Y 319.554,Z 381.677,A -85,B 0,C 180,E1 -15427.513,E2 -15427.513} C_VEL
LIN {X 0,Y 318.924,Z 381.76,A -85,B 0,C 180,E1 -15428.564,E2 -15428.564} C_VEL
LIN {X 0,Y 316.063,Z 382.116,A -85,B 0,C 180,E1 -15430.275,E2 -15430.275} C_VEL
LIN {X 0,Y 313.609,Z 382.417,A -85,B 0,C 180,E1 -15431.662,E2 -15431.662} C_VEL
LIN {X 0,Y 312.548,Z 382.551,A -85,B 0,C 180,E1 -15432.736,E2 -15432.736} C_VEL
LIN {X 0,Y 312.459,Z 382.557,A -85,B 0,C 180,E1 -15433.1,E2 -15433.1} C_VEL
LIN {X 0,Y 312.479,Z 382.557,A -85,B 0,C 180,E1 -15436.03,E2 -15436.03} C_VEL
LIN {X 0,Y 312.502,Z 382.555,A -85,B 0,C 180,E1 -15439.874,E2 -15439.874} C_VEL
LIN {X 0,Y 312.532,Z 382.551,A -85,B 0,C 180,E1 -15444.049,E2 -15444.049} C_VEL
LIN {X 0,Y 312.5,Z 382.557,A -85,B 0,C 180,E1 -15447.333,E2 -15447.333} C_VEL
LIN {X 0,Y 312.54,Z 382.552,A -85,B 0,C 180,E1 -15451.278,E2 -15451.278} C_VEL
LIN {X 0,Y 312.58,Z 382.55,A -85,B 0,C 180,E1 -15454.71,E2 -15454.71} C_VEL
LIN {X 0,Y 312.582,Z 382.545,A -85,B 0,C 180,E1 -15457.528,E2 -15457.528} C_VEL
LIN {X 0,Y 312.633,Z 382.538,A -85,B 0,C 180,E1 -15461.656,E2 -15461.656} C_VEL
LIN {X 0,Y 312.688,Z 382.532,A -85,B 0,C 180,E1 -15465.686,E2 -15465.686} C_VEL
LIN {X 0,Y 312.692,Z 382.53,A -85,B 0,C 180,E1 -15469.641,E2 -15469.641} C_VEL
LIN {X 0,Y 312.847,Z 382.513,A -85,B 0,C 180,E1 -15472.253,E2 -15472.253} C_VEL
LIN {X 0,Y 312.711,Z 382.532,A -85,B 0,C 180,E1 -15474.842,E2 -15474.842} C_VEL
LIN {X 0,Y 312.983,Z 382.495,A -85,B 0,C 180,E1 -15478.713,E2 -15478.713} C_VEL
LIN {X 0,Y 312.985,Z 382.487,A -85,B 0,C 180,E1 -15481.286,E2 -15481.286} C_VEL
LIN {X 0,Y 312.71,Z 382.528,A -85,B 0,C 180,E1 -15485.157,E2 -15485.157} C_VEL
LIN {X 0,Y 312.846,Z 382.513,A -85,B 0,C 180,E1 -15487.746,E2 -15487.746} C_VEL
LIN {X 0,Y 312.662,Z 382.534,A -85,B 0,C 180,E1 -15491.671,E2 -15491.671} C_VEL
LIN {X 0,Y 312.693,Z 382.533,A -85,B 0,C 180,E1 -15494.888,E2 -15494.888} C_VEL
LIN {X 0,Y 312.624,Z 382.54,A -85,B 0,C 180,E1 -15499.236,E2 -15499.236} C_VEL
LIN {X 0,Y 312.539,Z 382.551,A -85,B 0,C 180,E1 -15502.789,E2 -15502.789} C_VEL
LIN {X 0,Y 312.597,Z 382.547,A -85,B 0,C 180,E1 -15505.936,E2 -15505.936} C_VEL
LIN {X 0,Y 312.543,Z 382.552,A -85,B 0,C 180,E1 -15509.65,E2 -15509.65} C_VEL
LIN {X 0,Y 312.514,Z 382.556,A -85,B 0,C 180,E1 -15513.689,E2 -15513.689} C_VEL
LIN {X 0,Y 312.548,Z 382.551,A -85,B 0,C 180,E1 -15517.382,E2 -15517.382} C_VEL
LIN {X 0,Y 312.529,Z 382.554,A -85,B 0,C 180,E1 -15520.703,E2 -15520.703} C_VEL
LIN {X 0,Y 312.536,Z 382.556,A -85,B 0,C 180,E1 -15524.195,E2 -15524.195} C_VEL
LIN {X 0,Y 312.53,Z 382.557,A -85,B 0,C 180,E1 -15527.909,E2 -15527.909} C_VEL
LIN {X 0,Y 312.554,Z 382.555,A -85,B 0,C 180,E1 -15531.906,E2 -15531.906} C_VEL
LIN {X 0,Y 312.505,Z 382.56,A -85,B 0,C 180,E1 -15535.791,E2 -15535.791} C_VEL
LIN {X 0,Y 312.542,Z 382.689,A -85,B 0,C 180,E1 -15537.937,E2 -15537.937} C_VEL
LIN {X 0,Y 315.396,Z 395.905,A -85,B 0,C 180,E1 -15541.738,E2 -15541.738} C_VEL
LIN {X 0,Y 316.576,Z 402.834,A -85,B 0,C 180,E1 -15543.641,E2 -15543.641} C_VEL
LIN {X 0,Y 315.593,Z 411.815,A -85,B 0,C 180,E1 -15545.928,E2 -15545.928} C_VEL
LIN {X 0,Y 321.149,Z 454.916,A -85,B 0,C 180,E1 -15547.295,E2 -15547.295} C_VEL
LIN {X 0,Y 319.798,Z 520.449,A -85,B 0,C 180,E1 -15548.782,E2 -15548.782} C_VEL
LIN {X 0,Y 319.092,Z 533.729,A -85,B 0,C 180,E1 -15549.324,E2 -15549.324} C_VEL
LIN {X 0,Y 318.191,Z 545.936,A -85,B 0,C 180,E1 -15550.064,E2 -15550.064} C_VEL
LIN {X 0,Y 316.934,Z 558.229,A -85,B 0,C 180,E1 -15551.077,E2 -15551.077} C_VEL
LIN {X 0,Y 315.673,Z 569.889,A -85,B 0,C 180,E1 -15552.342,E2 -15552.342} C_VEL
LIN {X 0,Y 314.527,Z 580.147,A -85,B 0,C 180,E1 -15553.744,E2 -15553.744} C_VEL
LIN {X 0,Y 313.507,Z 589.827,A -85,B 0,C 180,E1 -15555.393,E2 -15555.393} C_VEL
LIN {X 0,Y 312.578,Z 597.561,A -85,B 0,C 180,E1 -15557.007,E2 -15557.007} C_VEL
LIN {X 0,Y 311.693,Z 605.125,A -85,B 0,C 180,E1 -15558.951,E2 -15558.951} C_VEL
LIN {X 0,Y 311.215,Z 611.203,A -85,B 0,C 180,E1 -15560.905,E2 -15560.905} C_VEL
LIN {X 0,Y 310.986,Z 615.998,A -85,B 0,C 180,E1 -15562.86,E2 -15562.86} C_VEL
LIN {X 0,Y 310.792,Z 619.639,A -85,B 0,C 180,E1 -15564.81,E2 -15564.81} C_VEL
LIN {X 0,Y 310.822,Z 621.514,A -85,B 0,C 180,E1 -15566.111,E2 -15566.111} C_VEL
LIN {X 0,Y 310.766,Z 622.906,A -85,B 0,C 180,E1 -15567.408,E2 -15567.408} C_VEL
LIN {X 0,Y 310.816,Z 623.893,A -85,B 0,C 180,E1 -15568.704,E2 -15568.704} C_VEL
LIN {X 0,Y 310.858,Z 624.484,A -85,B 0,C 180,E1 -15570,E2 -15570} C_VEL
LIN {X 0,Y 310.774,Z 624.67,A -85,B 0,C 180,E1 -15571.296,E2 -15571.296} C_VEL
LIN {X 0,Y 310.735,Z 624.423,A -85,B 0,C 180,E1 -15572.593,E2 -15572.593} C_VEL
LIN {X 0,Y 310.753,Z 623.786,A -85,B 0,C 180,E1 -15573.89,E2 -15573.89} C_VEL
LIN {X 0,Y 310.828,Z 621.337,A -85,B 0,C 180,E1 -15576.491,E2 -15576.491} C_VEL
LIN {X 0,Y 311.142,Z 618.372,A -85,B 0,C 180,E1 -15578.443,E2 -15578.443} C_VEL
LIN {X 0,Y 311.66,Z 614.389,A -85,B 0,C 180,E1 -15580.393,E2 -15580.393} C_VEL
LIN {X 0,Y 312.504,Z 609.297,A -85,B 0,C 180,E1 -15582.336,E2 -15582.336} C_VEL
LIN {X 0,Y 313.807,Z 602.931,A -85,B 0,C 180,E1 -15584.262,E2 -15584.262} C_VEL
LIN {X 0,Y 315.164,Z 595.347,A -85,B 0,C 180,E1 -15586.109,E2 -15586.109} C_VEL
LIN {X 0,Y 316.735,Z 586.978,A -85,B 0,C 180,E1 -15587.763,E2 -15587.763} C_VEL
LIN {X 0,Y 318.54,Z 577.21,A -85,B 0,C 180,E1 -15589.326,E2 -15589.326} C_VEL
LIN {X 0,Y 320.487,Z 566.352,A -85,B 0,C 180,E1 -15590.708,E2 -15590.708} C_VEL
LIN {X 0,Y 322.381,Z 554.002,A -85,B 0,C 180,E1 -15591.921,E2 -15591.921} C_VEL
LIN {X 0,Y 323.883,Z 541.937,A -85,B 0,C 180,E1 -15592.822,E2 -15592.822} C_VEL
LIN {X 0,Y 325.125,Z 529.46,A -85,B 0,C 180,E1 -15593.487,E2 -15593.487} C_VEL
LIN {X 0,Y 325.865,Z 516.606,A -85,B 0,C 180,E1 -15593.936,E2 -15593.936} C_VEL
LIN {X 0,Y 327.546,Z 455.528,A -85,B 0,C 180,E1 -15595.313,E2 -15595.313} C_VEL
LIN {X 0,Y 323.862,Z 432.908,A -85,B 0,C 180,E1 -15596.26,E2 -15596.26} C_VEL
LIN {X 0,Y 319.539,Z 412.949,A -85,B 0,C 180,E1 -15597.246,E2 -15597.246} C_VEL
LIN {X 0,Y 318.903,Z 410.623,A -85,B 0,C 180,E1 -15597.422,E2 -15597.422} C_VEL
LIN {X 0,Y 317.598,Z 403.317,A -85,B 0,C 180,E1 -15599.647,E2 -15599.647} C_VEL
LIN {X 0,Y 315.123,Z 392.662,A -85,B 0,C 180,E1 -15603.12,E2 -15603.12} C_VEL
LIN {X 0,Y 312.957,Z 384.243,A -85,B 0,C 180,E1 -15606.056,E2 -15606.056} C_VEL
LIN {X 0,Y 312.506,Z 382.56,A -85,B 0,C 180,E1 -15606.705,E2 -15606.705} C_VEL
LIN {X 0,Y 312.509,Z 382.561,A -85,B 0,C 180,E1 -15610.126,E2 -15610.126} C_VEL
LIN {X 0,Y 312.53,Z 382.557,A -85,B 0,C 180,E1 -15613.979,E2 -15613.979} C_VEL
LIN {X 0,Y 312.545,Z 382.551,A -85,B 0,C 180,E1 -15617.905,E2 -15617.905} C_VEL
LIN {X 0,Y 312.553,Z 382.553,A -85,B 0,C 180,E1 -15621.904,E2 -15621.904} C_VEL
LIN {X 0,Y 312.501,Z 382.554,A -85,B 0,C 180,E1 -15625.789,E2 -15625.789} C_VEL
LIN {X 0,Y 312.518,Z 382.554,A -85,B 0,C 180,E1 -15628.853,E2 -15628.853} C_VEL
LIN {X 0,Y 312.577,Z 382.55,A -85,B 0,C 180,E1 -15631.825,E2 -15631.825} C_VEL
LIN {X 0,Y 312.579,Z 382.542,A -85,B 0,C 180,E1 -15634.711,E2 -15634.711} C_VEL
LIN {X 0,Y 312.581,Z 382.541,A -85,B 0,C 180,E1 -15637.529,E2 -15637.529} C_VEL
LIN {X 0,Y 312.632,Z 382.537,A -85,B 0,C 180,E1 -15641.656,E2 -15641.656} C_VEL
LIN {X 0,Y 312.687,Z 382.535,A -85,B 0,C 180,E1 -15645.686,E2 -15645.686} C_VEL
LIN {X 0,Y 312.694,Z 382.536,A -85,B 0,C 180,E1 -15649.642,E2 -15649.642} C_VEL
LIN {X 0,Y 312.859,Z 382.501,A -85,B 0,C 180,E1 -15652.254,E2 -15652.254} C_VEL
LIN {X 0,Y 312.711,Z 382.532,A -85,B 0,C 180,E1 -15654.843,E2 -15654.843} C_VEL
LIN {X 0,Y 312.986,Z 382.491,A -85,B 0,C 180,E1 -15658.714,E2 -15658.714} C_VEL
LIN {X 0,Y 313.114,Z 382.482,A -85,B 0,C 180,E1 -15660,E2 -15660} C_VEL
LIN {X 0,Y 312.932,Z 382.492,A -85,B 0,C 180,E1 -15662.575,E2 -15662.575} C_VEL
LIN {X 0,Y 312.879,Z 382.505,A -85,B 0,C 180,E1 -15666.623,E2 -15666.623} C_VEL
LIN {X 0,Y 312.761,Z 382.524,A -85,B 0,C 180,E1 -15669.05,E2 -15669.05} C_VEL
LIN {X 0,Y 312.628,Z 382.536,A -85,B 0,C 180,E1 -15672.992,E2 -15672.992} C_VEL
LIN {X 0,Y 312.633,Z 382.534,A -85,B 0,C 180,E1 -15675.65,E2 -15675.65} C_VEL
LIN {X 0,Y 312.605,Z 382.539,A -85,B 0,C 180,E1 -15679.709,E2 -15679.709} C_VEL
LIN {X 0,Y 312.542,Z 382.554,A -85,B 0,C 180,E1 -15682.79,E2 -15682.79} C_VEL
LIN {X 0,Y 312.598,Z 382.546,A -85,B 0,C 180,E1 -15685.936,E2 -15685.936} C_VEL
LIN {X 0,Y 312.534,Z 382.552,A -85,B 0,C 180,E1 -15689.652,E2 -15689.652} C_VEL
LIN {X 0,Y 312.516,Z 382.542,A -85,B 0,C 180,E1 -15693.69,E2 -15693.69} C_VEL
LIN {X 0,Y 312.538,Z 382.553,A -85,B 0,C 180,E1 -15697.384,E2 -15697.384} C_VEL
LIN {X 0,Y 312.524,Z 382.558,A -85,B 0,C 180,E1 -15700.705,E2 -15700.705} C_VEL
LIN {X 0,Y 312.549,Z 382.615,A -85,B 0,C 180,E1 -15704.475,E2 -15704.475} C_VEL
LIN {X 0,Y 313.49,Z 386.636,A -85,B 0,C 180,E1 -15706.048,E2 -15706.048} C_VEL
LIN {X 0,Y 322.581,Z 404.679,A -85,B 0,C 180,E1 -15707.564,E2 -15707.564} C_VEL
LIN {X 0,Y 328.649,Z 418.68,A -85,B 0,C 180,E1 -15708.562,E2 -15708.562} C_VEL
LIN {X 0,Y 326.413,Z 492.34,A -85,B 0,C 180,E1 -15710.219,E2 -15710.219} C_VEL
LIN {X 0,Y 325.62,Z 506.03,A -85,B 0,C 180,E1 -15710.785,E2 -15710.785} C_VEL
LIN {X 0,Y 324.572,Z 517.813,A -85,B 0,C 180,E1 -15711.5,E2 -15711.5} C_VEL
LIN {X 0,Y 323.195,Z 529.881,A -85,B 0,C 180,E1 -15712.493,E2 -15712.493} C_VEL
LIN {X 0,Y 321.64,Z 540.731,A -85,B 0,C 180,E1 -15713.653,E2 -15713.653} C_VEL
LIN {X 0,Y 319.856,Z 551.858,A -85,B 0,C 180,E1 -15715.161,E2 -15715.161} C_VEL
LIN {X 0,Y 318.173,Z 561.084,A -85,B 0,C 180,E1 -15716.729,E2 -15716.729} C_VEL
LIN {X 0,Y 316.476,Z 569.639,A -85,B 0,C 180,E1 -15718.543,E2 -15718.543} C_VEL
LIN {X 0,Y 314.833,Z 577.337,A -85,B 0,C 180,E1 -15720.588,E2 -15720.588} C_VEL
LIN {X 0,Y 313.551,Z 583.391,A -85,B 0,C 180,E1 -15722.646,E2 -15722.646} C_VEL
LIN {X 0,Y 312.554,Z 588.044,A -85,B 0,C 180,E1 -15724.709,E2 -15724.709} C_VEL
LIN {X 0,Y 311.985,Z 590.463,A -85,B 0,C 180,E1 -15726.079,E2 -15726.079} C_VEL
LIN {X 0,Y 311.542,Z 592.65,A -85,B 0,C 180,E1 -15727.657,E2 -15727.657} C_VEL
LIN {X 0,Y 310.962,Z 594.839,A -85,B 0,C 180,E1 -15730.184,E2 -15730.184} C_VEL
LIN {X 0,Y 310.769,Z 595.469,A -85,B 0,C 180,E1 -15731.775,E2 -15731.775} C_VEL
LIN {X 0,Y 310.64,Z 595.23,A -85,B 0,C 180,E1 -15734.247,E2 -15734.247} C_VEL
LIN {X 0,Y 310.713,Z 593.729,A -85,B 0,C 180,E1 -15736.563,E2 -15736.563} C_VEL
LIN {X 0,Y 310.996,Z 590.869,A -85,B 0,C 180,E1 -15738.926,E2 -15738.926} C_VEL
LIN {X 0,Y 311.349,Z 587.323,A -85,B 0,C 180,E1 -15740.909,E2 -15740.909} C_VEL
LIN {X 0,Y 311.866,Z 582.504,A -85,B 0,C 180,E1 -15742.936,E2 -15742.936} C_VEL
LIN {X 0,Y 312.604,Z 575.619,A -85,B 0,C 180,E1 -15745.164,E2 -15745.164} C_VEL
LIN {X 0,Y 313.541,Z 567.998,A -85,B 0,C 180,E1 -15747.109,E2 -15747.109} C_VEL
LIN {X 0,Y 314.47,Z 560.206,A -85,B 0,C 180,E1 -15748.719,E2 -15748.719} C_VEL
LIN {X 0,Y 315.773,Z 549.583,A -85,B 0,C 180,E1 -15750.479,E2 -15750.479} C_VEL
LIN {X 0,Y 316.845,Z 539.694,A -85,B 0,C 180,E1 -15751.796,E2 -15751.796} C_VEL
LIN {X 0,Y 317.926,Z 528.289,A -85,B 0,C 180,E1 -15753.009,E2 -15753.009} C_VEL
LIN {X 0,Y 318.964,Z 515.629,A -85,B 0,C 180,E1 -15754.027,E2 -15754.027} C_VEL
LIN {X 0,Y 319.702,Z 503.028,A -85,B 0,C 180,E1 -15754.768,E2 -15754.768} C_VEL
LIN {X 0,Y 320.146,Z 490.992,A -85,B 0,C 180,E1 -15755.241,E2 -15755.241} C_VEL
LIN {X 0,Y 321.746,Z 412.308,A -85,B 0,C 180,E1 -15757.013,E2 -15757.013} C_VEL
LIN {X 0,Y 320.231,Z 405.912,A -85,B 0,C 180,E1 -15757.258,E2 -15757.258} C_VEL
LIN {X 0,Y 314.109,Z 387.576,A -85,B 0,C 180,E1 -15758.092,E2 -15758.092} C_VEL
LIN {X 0,Y 313.334,Z 385.233,A -85,B 0,C 180,E1 -15758.201,E2 -15758.201} C_VEL
LIN {X 0,Y 312.759,Z 382.529,A -85,B 0,C 180,E1 -15759.131,E2 -15759.131} C_VEL
LIN {X 0,Y 312.639,Z 382.543,A -85,B 0,C 180,E1 -15762.991,E2 -15762.991} C_VEL
LIN {X 0,Y 312.642,Z 382.542,A -85,B 0,C 180,E1 -15765.649,E2 -15765.649} C_VEL
LIN {X 0,Y 312.634,Z 382.544,A -85,B 0,C 180,E1 -15769.236,E2 -15769.236} C_VEL
LIN {X 0,Y 312.549,Z 382.551,A -85,B 0,C 180,E1 -15772.789,E2 -15772.789} C_VEL
LIN {X 0,Y 312.605,Z 382.543,A -85,B 0,C 180,E1 -15775.935,E2 -15775.935} C_VEL
LIN {X 0,Y 312.547,Z 382.552,A -85,B 0,C 180,E1 -15779.649,E2 -15779.649} C_VEL
LIN {X 0,Y 312.521,Z 382.555,A -85,B 0,C 180,E1 -15783.688,E2 -15783.688} C_VEL
LIN {X 0,Y 312.52,Z 382.555,A -85,B 0,C 180,E1 -15787.501,E2 -15787.501} C_VEL
LIN {X 0,Y 312.49,Z 382.559,A -85,B 0,C 180,E1 -15790.708,E2 -15790.708} C_VEL
LIN {X 0,Y 312.459,Z 382.557,A -85,B 0,C 180,E1 -15793.1,E2 -15793.1} C_VEL
LIN {X 0,Y 311.784,Z 382.646,A -85,B 0,C 180,E1 -15794.176,E2 -15794.176} C_VEL
LIN {X 0,Y 308.93,Z 382.999,A -85,B 0,C 180,E1 -15795.928,E2 -15795.928} C_VEL
LIN {X 0,Y 306.524,Z 383.301,A -85,B 0,C 180,E1 -15797.349,E2 -15797.349} C_VEL
LIN {X 0,Y 305.505,Z 383.427,A -85,B 0,C 180,E1 -15798.449,E2 -15798.449} C_VEL
LIN {X 0,Y 305.429,Z 383.435,A -85,B 0,C 180,E1 -15798.821,E2 -15798.821} C_VEL
LIN {X 0,Y 305.465,Z 383.431,A -85,B 0,C 180,E1 -15801.595,E2 -15801.595} C_VEL
LIN {X 0,Y 305.459,Z 383.437,A -85,B 0,C 180,E1 -15804.886,E2 -15804.886} C_VEL
LIN {X 0,Y 305.446,Z 383.435,A -85,B 0,C 180,E1 -15808.355,E2 -15808.355} C_VEL
LIN {X 0,Y 305.509,Z 383.429,A -85,B 0,C 180,E1 -15811.112,E2 -15811.112} C_VEL
LIN {X 0,Y 305.561,Z 383.42,A -85,B 0,C 180,E1 -15814.086,E2 -15814.086} C_VEL
LIN {X 0,Y 305.496,Z 383.429,A -85,B 0,C 180,E1 -15818.402,E2 -15818.402} C_VEL
LIN {X 0,Y 305.585,Z 383.418,A -85,B 0,C 180,E1 -15821.217,E2 -15821.217} C_VEL
LIN {X 0,Y 305.643,Z 383.41,A -85,B 0,C 180,E1 -15825.348,E2 -15825.348} C_VEL
LIN {X 0,Y 305.629,Z 383.41,A -85,B 0,C 180,E1 -15829.399,E2 -15829.399} C_VEL
LIN {X 0,Y 305.79,Z 383.391,A -85,B 0,C 180,E1 -15832.073,E2 -15832.073} C_VEL
LIN {X 0,Y 305.682,Z 383.409,A -85,B 0,C 180,E1 -15834.723,E2 -15834.723} C_VEL
LIN {X 0,Y 305.95,Z 383.37,A -85,B 0,C 180,E1 -15838.683,E2 -15838.683} C_VEL
LIN {X 0,Y 305.952,Z 383.362,A -85,B 0,C 180,E1 -15841.316,E2 -15841.316} C_VEL
LIN {X 0,Y 305.681,Z 383.403,A -85,B 0,C 180,E1 -15845.276,E2 -15845.276} C_VEL
LIN {X 0,Y 305.79,Z 383.393,A -85,B 0,C 180,E1 -15847.926,E2 -15847.926} C_VEL
LIN {X 0,Y 305.596,Z 383.416,A -85,B 0,C 180,E1 -15851.945,E2 -15851.945} C_VEL
LIN {X 0,Y 305.631,Z 383.412,A -85,B 0,C 180,E1 -15855.035,E2 -15855.035} C_VEL
LIN {X 0,Y 305.57,Z 383.418,A -85,B 0,C 180,E1 -15859.445,E2 -15859.445} C_VEL
LIN {X 0,Y 305.484,Z 383.429,A -85,B 0,C 180,E1 -15863.041,E2 -15863.041} C_VEL
LIN {X 0,Y 305.542,Z 383.428,A -85,B 0,C 180,E1 -15866.227,E2 -15866.227} C_VEL
LIN {X 0,Y 305.497,Z 383.429,A -85,B 0,C 180,E1 -15869.053,E2 -15869.053} C_VEL
LIN {X 0,Y 305.46,Z 383.434,A -85,B 0,C 180,E1 -15873.517,E2 -15873.517} C_VEL
LIN {X 0,Y 305.498,Z 383.43,A -85,B 0,C 180,E1 -15876.736,E2 -15876.736} C_VEL
LIN {X 0,Y 305.49,Z 383.432,A -85,B 0,C 180,E1 -15880.609,E2 -15880.609} C_VEL
LIN {X 0,Y 305.493,Z 383.432,A -85,B 0,C 180,E1 -15883.643,E2 -15883.643} C_VEL
LIN {X 0,Y 305.495,Z 383.43,A -85,B 0,C 180,E1 -15887.406,E2 -15887.406} C_VEL
LIN {X 0,Y 305.515,Z 383.429,A -85,B 0,C 180,E1 -15891.604,E2 -15891.604} C_VEL
LIN {X 0,Y 305.461,Z 383.435,A -85,B 0,C 180,E1 -15894.888,E2 -15894.888} C_VEL
LIN {X 0,Y 305.497,Z 383.48,A -85,B 0,C 180,E1 -15897.568,E2 -15897.568} C_VEL
LIN {X 0,Y 308.285,Z 396.468,A -85,B 0,C 180,E1 -15901.398,E2 -15901.398} C_VEL
LIN {X 0,Y 309.602,Z 404.761,A -85,B 0,C 180,E1 -15903.727,E2 -15903.727} C_VEL
LIN {X 0,Y 308.754,Z 411.446,A -85,B 0,C 180,E1 -15905.465,E2 -15905.465} C_VEL
LIN {X 0,Y 314.4,Z 455.496,A -85,B 0,C 180,E1 -15906.91,E2 -15906.91} C_VEL
LIN {X 0,Y 313.041,Z 519.632,A -85,B 0,C 180,E1 -15908.388,E2 -15908.388} C_VEL
LIN {X 0,Y 312.318,Z 533.094,A -85,B 0,C 180,E1 -15908.941,E2 -15908.941} C_VEL
LIN {X 0,Y 311.296,Z 546.52,A -85,B 0,C 180,E1 -15909.776,E2 -15909.776} C_VEL
LIN {X 0,Y 310,Z 558.546,A -85,B 0,C 180,E1 -15910.809,E2 -15910.809} C_VEL
LIN {X 0,Y 308.711,Z 570.091,A -85,B 0,C 180,E1 -15912.102,E2 -15912.102} C_VEL
LIN {X 0,Y 307.568,Z 579.852,A -85,B 0,C 180,E1 -15913.472,E2 -15913.472} C_VEL
LIN {X 0,Y 306.607,Z 589.006,A -85,B 0,C 180,E1 -15915.057,E2 -15915.057} C_VEL
LIN {X 0,Y 305.439,Z 598.196,A -85,B 0,C 180,E1 -15917.036,E2 -15917.036} C_VEL
LIN {X 0,Y 304.577,Z 605.592,A -85,B 0,C 180,E1 -15919.026,E2 -15919.026} C_VEL
LIN {X 0,Y 304.172,Z 610.6,A -85,B 0,C 180,E1 -15920.692,E2 -15920.692} C_VEL
LIN {X 0,Y 303.915,Z 615.452,A -85,B 0,C 180,E1 -15922.693,E2 -15922.693} C_VEL
LIN {X 0,Y 303.705,Z 619.147,A -85,B 0,C 180,E1 -15924.689,E2 -15924.689} C_VEL
